LIN {X 0,Y 566.18,Z 159.454,A -85,B 0,C 180,E1 -2663.788,E2 -2663.788} C_VEL
LIN {X 0,Y 566.208,Z 159.454,A -85,B 0,C 180,E1 -2666.265,E2 -2666.265} C_VEL
LIN {X 0,Y 566.189,Z 159.457,A -85,B 0,C 180,E1 -2668.923,E2 -2668.923} C_VEL
LIN {X 0,Y 566.207,Z 159.451,A -85,B 0,C 180,E1 -2671.857,E2 -2671.857} C_VEL
LIN {X 0,Y 566.205,Z 159.457,A -85,B 0,C 180,E1 -2674.25,E2 -2674.25} C_VEL
LIN {X 0,Y 566.186,Z 159.457,A -85,B 0,C 180,E1 -2676.713,E2 -2676.713} C_VEL
LIN {X 0,Y 566.207,Z 159.452,A -85,B 0,C 180,E1 -2679.662,E2 -2679.662} C_VEL
LIN {X 0,Y 566.194,Z 159.455,A -85,B 0,C 180,E1 -2682.668,E2 -2682.668} C_VEL
LIN {X 0,Y 566.228,Z 159.45,A -85,B 0,C 180,E1 -2685.626,E2 -2685.626} C_VEL
LIN {X 0,Y 566.229,Z 159.449,A -85,B 0,C 180,E1 -2688.675,E2 -2688.675} C_VEL
LIN {X 0,Y 566.228,Z 159.45,A -85,B 0,C 180,E1 -2691.434,E2 -2691.434} C_VEL
LIN {X 0,Y 566.248,Z 159.448,A -85,B 0,C 180,E1 -2694.301,E2 -2694.301} C_VEL
LIN {X 0,Y 566.27,Z 159.45,A -85,B 0,C 180,E1 -2697.866,E2 -2697.866} C_VEL
LIN {X 0,Y 566.295,Z 159.439,A -85,B 0,C 180,E1 -2700.711,E2 -2700.711} C_VEL
LIN {X 0,Y 566.266,Z 159.444,A -85,B 0,C 180,E1 -2702.845,E2 -2702.845} C_VEL
LIN {X 0,Y 566.252,Z 159.451,A -85,B 0,C 180,E1 -2705.698,E2 -2705.698} C_VEL
LIN {X 0,Y 566.226,Z 159.448,A -85,B 0,C 180,E1 -2708.565,E2 -2708.565} C_VEL
LIN {X 0,Y 566.235,Z 159.455,A -85,B 0,C 180,E1 -2711.454,E2 -2711.454} C_VEL
LIN {X 0,Y 566.227,Z 159.449,A -85,B 0,C 180,E1 -2714.506,E2 -2714.506} C_VEL
LIN {X 0,Y 566.193,Z 159.459,A -85,B 0,C 180,E1 -2717.331,E2 -2717.331} C_VEL
LIN {X 0,Y 566.212,Z 159.45,A -85,B 0,C 180,E1 -2720.337,E2 -2720.337} C_VEL
LIN {X 0,Y 566.182,Z 159.457,A -85,B 0,C 180,E1 -2723.404,E2 -2723.404} C_VEL
LIN {X 0,Y 566.206,Z 159.451,A -85,B 0,C 180,E1 -2725.749,E2 -2725.749} C_VEL
LIN {X 0,Y 566.205,Z 159.452,A -85,B 0,C 180,E1 -2727.482,E2 -2727.482} C_VEL
LIN {X 0,Y 565.53,Z 159.536,A -85,B 0,C 180,E1 -2728.076,E2 -2728.076} C_VEL
LIN {X 0,Y 562.668,Z 159.897,A -85,B 0,C 180,E1 -2729.039,E2 -2729.039} C_VEL
LIN {X 0,Y 560.256,Z 160.195,A -85,B 0,C 180,E1 -2729.815,E2 -2729.815} C_VEL
LIN {X 0,Y 559.225,Z 160.324,A -85,B 0,C 180,E1 -2730.414,E2 -2730.414} C_VEL
LIN {X 0,Y 559.143,Z 160.332,A -85,B 0,C 180,E1 -2730.617,E2 -2730.617} C_VEL
LIN {X 0,Y 559.158,Z 160.329,A -85,B 0,C 180,E1 -2733.575,E2 -2733.575} C_VEL
LIN {X 0,Y 559.162,Z 160.335,A -85,B 0,C 180,E1 -2736.449,E2 -2736.449} C_VEL
LIN {X 0,Y 559.172,Z 160.33,A -85,B 0,C 180,E1 -2738.934,E2 -2738.934} C_VEL
LIN {X 0,Y 559.186,Z 160.326,A -85,B 0,C 180,E1 -2741.768,E2 -2741.768} C_VEL
LIN {X 0,Y 559.133,Z 160.335,A -85,B 0,C 180,E1 -2744.739,E2 -2744.739} C_VEL
LIN {X 0,Y 559.155,Z 160.329,A -85,B 0,C 180,E1 -2747.257,E2 -2747.257} C_VEL
LIN {X 0,Y 559.18,Z 160.335,A -85,B 0,C 180,E1 -2750.135,E2 -2750.135} C_VEL
LIN {X 0,Y 559.141,Z 160.331,A -85,B 0,C 180,E1 -2752.892,E2 -2752.892} C_VEL
LIN {X 0,Y 559.152,Z 160.332,A -85,B 0,C 180,E1 -2755.556,E2 -2755.556} C_VEL
LIN {X 0,Y 559.166,Z 160.334,A -85,B 0,C 180,E1 -2758.138,E2 -2758.138} C_VEL
LIN {X 0,Y 559.152,Z 160.33,A -85,B 0,C 180,E1 -2760.647,E2 -2760.647} C_VEL
LIN {X 0,Y 559.167,Z 160.329,A -85,B 0,C 180,E1 -2763.172,E2 -2763.172} C_VEL
LIN {X 0,Y 559.153,Z 160.335,A -85,B 0,C 180,E1 -2765.495,E2 -2765.495} C_VEL
LIN {X 0,Y 559.168,Z 160.327,A -85,B 0,C 180,E1 -2768.624,E2 -2768.624} C_VEL
LIN {X 0,Y 559.165,Z 160.329,A -85,B 0,C 180,E1 -2770.926,E2 -2770.926} C_VEL
LIN {X 0,Y 559.164,Z 160.332,A -85,B 0,C 180,E1 -2773.948,E2 -2773.948} C_VEL
LIN {X 0,Y 559.17,Z 160.329,A -85,B 0,C 180,E1 -2776.184,E2 -2776.184} C_VEL
LIN {X 0,Y 559.193,Z 160.332,A -85,B 0,C 180,E1 -2779.134,E2 -2779.134} C_VEL
LIN {X 0,Y 559.203,Z 160.325,A -85,B 0,C 180,E1 -2782.054,E2 -2782.054} C_VEL
LIN {X 0,Y 559.253,Z 160.324,A -85,B 0,C 180,E1 -2784.953,E2 -2784.953} C_VEL
LIN {X 0,Y 559.254,Z 160.318,A -85,B 0,C 180,E1 -2787.839,E2 -2787.839} C_VEL
LIN {X 0,Y 559.27,Z 160.322,A -85,B 0,C 180,E1 -2790.72,E2 -2790.72} C_VEL
LIN {X 0,Y 559.236,Z 160.328,A -85,B 0,C 180,E1 -2792.881,E2 -2792.881} C_VEL
LIN {X 0,Y 559.235,Z 160.32,A -85,B 0,C 180,E1 -2795.77,E2 -2795.77} C_VEL
LIN {X 0,Y 559.189,Z 160.334,A -85,B 0,C 180,E1 -2798.674,E2 -2798.674} C_VEL
LIN {X 0,Y 559.202,Z 160.324,A -85,B 0,C 180,E1 -2801.6,E2 -2801.6} C_VEL
LIN {X 0,Y 559.196,Z 160.333,A -85,B 0,C 180,E1 -2804.595,E2 -2804.595} C_VEL
LIN {X 0,Y 559.156,Z 160.33,A -85,B 0,C 180,E1 -2807.557,E2 -2807.557} C_VEL
LIN {X 0,Y 559.169,Z 160.329,A -85,B 0,C 180,E1 -2809.837,E2 -2809.837} C_VEL
LIN {X 0,Y 559.138,Z 160.338,A -85,B 0,C 180,E1 -2812.153,E2 -2812.153} C_VEL
LIN {X 0,Y 559.175,Z 160.326,A -85,B 0,C 180,E1 -2815.187,E2 -2815.187} C_VEL
LIN {X 0,Y 559.188,Z 160.328,A -85,B 0,C 180,E1 -2817.711,E2 -2817.711} C_VEL
LIN {X 0,Y 559.164,Z 160.336,A -85,B 0,C 180,E1 -2820.182,E2 -2820.182} C_VEL
LIN {X 0,Y 559.17,Z 160.328,A -85,B 0,C 180,E1 -2822.714,E2 -2822.714} C_VEL
LIN {X 0,Y 559.153,Z 160.33,A -85,B 0,C 180,E1 -2825.322,E2 -2825.322} C_VEL
LIN {X 0,Y 559.13,Z 160.339,A -85,B 0,C 180,E1 -2828.017,E2 -2828.017} C_VEL
LIN {X 0,Y 559.171,Z 160.327,A -85,B 0,C 180,E1 -2830.81,E2 -2830.81} C_VEL
LIN {X 0,Y 559.153,Z 160.338,A -85,B 0,C 180,E1 -2833.732,E2 -2833.732} C_VEL
LIN {X 0,Y 559.143,Z 160.331,A -85,B 0,C 180,E1 -2836.803,E2 -2836.803} C_VEL
LIN {X 0,Y 559.17,Z 160.331,A -85,B 0,C 180,E1 -2839.189,E2 -2839.189} C_VEL
LIN {X 0,Y 559.128,Z 160.334,A -85,B 0,C 180,E1 -2841.983,E2 -2841.983} C_VEL
LIN {X 0,Y 559.153,Z 160.331,A -85,B 0,C 180,E1 -2844.783,E2 -2844.783} C_VEL
LIN {X 0,Y 559.167,Z 160.336,A -85,B 0,C 180,E1 -2847.361,E2 -2847.361} C_VEL
LIN {X 0,Y 559.182,Z 160.326,A -85,B 0,C 180,E1 -2850.135,E2 -2850.135} C_VEL
LIN {X 0,Y 559.164,Z 160.337,A -85,B 0,C 180,E1 -2853.172,E2 -2853.172} C_VEL
LIN {X 0,Y 559.15,Z 160.333,A -85,B 0,C 180,E1 -2855.495,E2 -2855.495} C_VEL
LIN {X 0,Y 559.17,Z 160.331,A -85,B 0,C 180,E1 -2858.624,E2 -2858.624} C_VEL
LIN {X 0,Y 559.162,Z 160.337,A -85,B 0,C 180,E1 -2860.926,E2 -2860.926} C_VEL
LIN {X 0,Y 559.164,Z 160.328,A -85,B 0,C 180,E1 -2863.948,E2 -2863.948} C_VEL
LIN {X 0,Y 559.168,Z 160.329,A -85,B 0,C 180,E1 -2866.184,E2 -2866.184} C_VEL
LIN {X 0,Y 559.188,Z 160.327,A -85,B 0,C 180,E1 -2869.134,E2 -2869.134} C_VEL
LIN {X 0,Y 559.2,Z 160.326,A -85,B 0,C 180,E1 -2872.054,E2 -2872.054} C_VEL
LIN {X 0,Y 559.247,Z 160.32,A -85,B 0,C 180,E1 -2874.954,E2 -2874.954} C_VEL
LIN {X 0,Y 559.241,Z 160.32,A -85,B 0,C 180,E1 -2877.84,E2 -2877.84} C_VEL
LIN {X 0,Y 559.27,Z 160.318,A -85,B 0,C 180,E1 -2880.72,E2 -2880.72} C_VEL
LIN {X 0,Y 559.234,Z 160.32,A -85,B 0,C 180,E1 -2882.882,E2 -2882.882} C_VEL
LIN {X 0,Y 559.218,Z 160.325,A -85,B 0,C 180,E1 -2885.771,E2 -2885.771} C_VEL
LIN {X 0,Y 559.186,Z 160.326,A -85,B 0,C 180,E1 -2888.675,E2 -2888.675} C_VEL
LIN {X 0,Y 559.199,Z 160.327,A -85,B 0,C 180,E1 -2891.601,E2 -2891.601} C_VEL
LIN {X 0,Y 559.194,Z 160.325,A -85,B 0,C 180,E1 -2894.596,E2 -2894.596} C_VEL
LIN {X 0,Y 559.153,Z 160.335,A -85,B 0,C 180,E1 -2897.557,E2 -2897.557} C_VEL
LIN {X 0,Y 559.164,Z 160.335,A -85,B 0,C 180,E1 -2899.838,E2 -2899.838} C_VEL
LIN {X 0,Y 559.136,Z 160.334,A -85,B 0,C 180,E1 -2902.153,E2 -2902.153} C_VEL
LIN {X 0,Y 559.17,Z 160.332,A -85,B 0,C 180,E1 -2905.299,E2 -2905.299} C_VEL
LIN {X 0,Y 559.145,Z 160.336,A -85,B 0,C 180,E1 -2907.714,E2 -2907.714} C_VEL
LIN {X 0,Y 559.15,Z 160.33,A -85,B 0,C 180,E1 -2910.183,E2 -2910.183} C_VEL
LIN {X 0,Y 559.152,Z 160.331,A -85,B 0,C 180,E1 -2912.716,E2 -2912.716} C_VEL
LIN {X 0,Y 559.123,Z 160.342,A -85,B 0,C 180,E1 -2915.325,E2 -2915.325} C_VEL
LIN {X 0,Y 559.129,Z 160.334,A -85,B 0,C 180,E1 -2918.018,E2 -2918.018} C_VEL
LIN {X 0,Y 559.152,Z 160.336,A -85,B 0,C 180,E1 -2920.813,E2 -2920.813} C_VEL
LIN {X 0,Y 559.134,Z 160.336,A -85,B 0,C 180,E1 -2923.735,E2 -2923.735} C_VEL
LIN {X 0,Y 559.119,Z 160.342,A -85,B 0,C 180,E1 -2926.265,E2 -2926.265} C_VEL
LIN {X 0,Y 559.534,Z 163.189,A -85,B 0,C 180,E1 -2928.264,E2 -2928.264} C_VEL
LIN {X 0,Y 559.526,Z 166.347,A -85,B 0,C 180,E1 -2930.165,E2 -2930.165} C_VEL
LIN {X 0,Y 559.373,Z 171.292,A -85,B 0,C 180,E1 -2932.91,E2 -2932.91} C_VEL
LIN {X 0,Y 559.267,Z 176.344,A -85,B 0,C 180,E1 -2935.564,E2 -2935.564} C_VEL
LIN {X 0,Y 559.205,Z 181.734,A -85,B 0,C 180,E1 -2938.14,E2 -2938.14} C_VEL
LIN {X 0,Y 559.124,Z 187.123,A -85,B 0,C 180,E1 -2940.646,E2 -2940.646} C_VEL
LIN {X 0,Y 559.091,Z 192.725,A -85,B 0,C 180,E1 -2943.189,E2 -2943.189} C_VEL
LIN {X 0,Y 559.021,Z 197.902,A -85,B 0,C 180,E1 -2945.489,E2 -2945.489} C_VEL
LIN {X 0,Y 559.005,Z 204.794,A -85,B 0,C 180,E1 -2948.491,E2 -2948.491} C_VEL
LIN {X 0,Y 558.93,Z 210.478,A -85,B 0,C 180,E1 -2950.918,E2 -2950.918} C_VEL
LIN {X 0,Y 558.881,Z 215.868,A -85,B 0,C 180,E1 -2953.189,E2 -2953.189} C_VEL
LIN {X 0,Y 558.834,Z 223.054,A -85,B 0,C 180,E1 -2956.176,E2 -2956.176} C_VEL
LIN {X 0,Y 558.829,Z 225.524,A -85,B 0,C 180,E1 -2957.194,E2 -2957.194} C_VEL
LIN {X 0,Y 559.988,Z 233.412,A -85,B 0,C 180,E1 -2957.382,E2 -2957.382} C_VEL
LIN {X 0,Y 559.865,Z 245.248,A -85,B 0,C 180,E1 -2957.729,E2 -2957.729} C_VEL
LIN {X 0,Y 559.716,Z 256.248,A -85,B 0,C 180,E1 -2958.171,E2 -2958.171} C_VEL
LIN {X 0,Y 559.532,Z 267.866,A -85,B 0,C 180,E1 -2958.779,E2 -2958.779} C_VEL
LIN {X 0,Y 559.42,Z 279.921,A -85,B 0,C 180,E1 -2959.596,E2 -2959.596} C_VEL
LIN {X 0,Y 559.242,Z 289.58,A -85,B 0,C 180,E1 -2960.415,E2 -2960.415} C_VEL
LIN {X 0,Y 559.127,Z 298.385,A -85,B 0,C 180,E1 -2961.325,E2 -2961.325} C_VEL
LIN {X 0,Y 558.996,Z 307.008,A -85,B 0,C 180,E1 -2962.414,E2 -2962.414} C_VEL
LIN {X 0,Y 558.894,Z 313.872,A -85,B 0,C 180,E1 -2963.502,E2 -2963.502} C_VEL
LIN {X 0,Y 558.868,Z 319.364,A -85,B 0,C 180,E1 -2964.588,E2 -2964.588} C_VEL
LIN {X 0,Y 558.869,Z 323.664,A -85,B 0,C 180,E1 -2965.673,E2 -2965.673} C_VEL
LIN {X 0,Y 558.836,Z 325.966,A -85,B 0,C 180,E1 -2966.395,E2 -2966.395} C_VEL
LIN {X 0,Y 558.799,Z 327.792,A -85,B 0,C 180,E1 -2967.116,E2 -2967.116} C_VEL
LIN {X 0,Y 558.745,Z 330.19,A -85,B 0,C 180,E1 -2968.559,E2 -2968.559} C_VEL
LIN {X 0,Y 558.741,Z 330.782,A -85,B 0,C 180,E1 -2969.279,E2 -2969.279} C_VEL
LIN {X 0,Y 558.741,Z 330.782,A -85,B 0,C 180,E1 -2970.721,E2 -2970.721} C_VEL
LIN {X 0,Y 558.745,Z 330.19,A -85,B 0,C 180,E1 -2971.441,E2 -2971.441} C_VEL
LIN {X 0,Y 558.799,Z 327.792,A -85,B 0,C 180,E1 -2972.884,E2 -2972.884} C_VEL
LIN {X 0,Y 558.844,Z 324.879,A -85,B 0,C 180,E1 -2973.966,E2 -2973.966} C_VEL
LIN {X 0,Y 558.798,Z 320.93,A -85,B 0,C 180,E1 -2975.051,E2 -2975.051} C_VEL
LIN {X 0,Y 558.909,Z 315.835,A -85,B 0,C 180,E1 -2976.136,E2 -2976.136} C_VEL
LIN {X 0,Y 558.974,Z 309.452,A -85,B 0,C 180,E1 -2977.223,E2 -2977.223} C_VEL
LIN {X 0,Y 559.099,Z 301.491,A -85,B 0,C 180,E1 -2978.312,E2 -2978.312} C_VEL
LIN {X 0,Y 559.207,Z 293.35,A -85,B 0,C 180,E1 -2979.221,E2 -2979.221} C_VEL
LIN {X 0,Y 559.346,Z 283.358,A -85,B 0,C 180,E1 -2980.131,E2 -2980.131} C_VEL
LIN {X 0,Y 559.457,Z 273.539,A -85,B 0,C 180,E1 -2980.861,E2 -2980.861} C_VEL
LIN {X 0,Y 559.608,Z 262.505,A -85,B 0,C 180,E1 -2981.523,E2 -2981.523} C_VEL
LIN {X 0,Y 559.807,Z 248.984,A -85,B 0,C 180,E1 -2982.139,E2 -2982.139} C_VEL
LIN {X 0,Y 559.952,Z 236.981,A -85,B 0,C 180,E1 -2982.527,E2 -2982.527} C_VEL
LIN {X 0,Y 559.759,Z 231.126,A -85,B 0,C 180,E1 -2982.678,E2 -2982.678} C_VEL
LIN {X 0,Y 558.829,Z 225.524,A -85,B 0,C 180,E1 -2982.806,E2 -2982.806} C_VEL
LIN {X 0,Y 558.857,Z 219.461,A -85,B 0,C 180,E1 -2985.313,E2 -2985.313} C_VEL
LIN {X 0,Y 558.904,Z 212.275,A -85,B 0,C 180,E1 -2988.322,E2 -2988.322} C_VEL
LIN {X 0,Y 558.945,Z 206.885,A -85,B 0,C 180,E1 -2990.613,E2 -2990.613} C_VEL
LIN {X 0,Y 559.028,Z 200.432,A -85,B 0,C 180,E1 -2993.401,E2 -2993.401} C_VEL
LIN {X 0,Y 559.068,Z 194.309,A -85,B 0,C 180,E1 -2996.102,E2 -2996.102} C_VEL
LIN {X 0,Y 559.11,Z 188.92,A -85,B 0,C 180,E1 -2998.532,E2 -2998.532} C_VEL
LIN {X 0,Y 559.183,Z 182.972,A -85,B 0,C 180,E1 -3001.279,E2 -3001.279} C_VEL
LIN {X 0,Y 559.26,Z 177.321,A -85,B 0,C 180,E1 -3003.963,E2 -3003.963} C_VEL
LIN {X 0,Y 559.361,Z 172.43,A -85,B 0,C 180,E1 -3006.474,E2 -3006.474} C_VEL
LIN {X 0,Y 559.508,Z 167.979,A -85,B 0,C 180,E1 -3008.906,E2 -3008.906} C_VEL
LIN {X 0,Y 559.596,Z 164.18,A -85,B 0,C 180,E1 -3011.101,E2 -3011.101} C_VEL
LIN {X 0,Y 559.206,Z 160.915,A -85,B 0,C 180,E1 -3013.203,E2 -3013.203} C_VEL
LIN {X 0,Y 559.119,Z 160.34,A -85,B 0,C 180,E1 -3013.735,E2 -3013.735} C_VEL
LIN {X 0,Y 559.134,Z 160.335,A -85,B 0,C 180,E1 -3016.265,E2 -3016.265} C_VEL
LIN {X 0,Y 559.152,Z 160.336,A -85,B 0,C 180,E1 -3019.187,E2 -3019.187} C_VEL
LIN {X 0,Y 559.129,Z 160.334,A -85,B 0,C 180,E1 -3021.982,E2 -3021.982} C_VEL
LIN {X 0,Y 559.127,Z 160.342,A -85,B 0,C 180,E1 -3024.787,E2 -3024.787} C_VEL
LIN {X 0,Y 559.152,Z 160.33,A -85,B 0,C 180,E1 -3027.364,E2 -3027.364} C_VEL
LIN {X 0,Y 559.144,Z 160.333,A -85,B 0,C 180,E1 -3030.142,E2 -3030.142} C_VEL
LIN {X 0,Y 559.161,Z 160.329,A -85,B 0,C 180,E1 -3033.173,E2 -3033.173} C_VEL
LIN {X 0,Y 559.153,Z 160.329,A -85,B 0,C 180,E1 -3035.494,E2 -3035.494} C_VEL
LIN {X 0,Y 559.167,Z 160.332,A -85,B 0,C 180,E1 -3038.623,E2 -3038.623} C_VEL
LIN {X 0,Y 559.157,Z 160.33,A -85,B 0,C 180,E1 -3040.925,E2 -3040.925} C_VEL
LIN {X 0,Y 559.162,Z 160.334,A -85,B 0,C 180,E1 -3043.947,E2 -3043.947} C_VEL
LIN {X 0,Y 559.166,Z 160.336,A -85,B 0,C 180,E1 -3046.184,E2 -3046.184} C_VEL
LIN {X 0,Y 559.19,Z 160.325,A -85,B 0,C 180,E1 -3049.133,E2 -3049.133} C_VEL
LIN {X 0,Y 559.196,Z 160.331,A -85,B 0,C 180,E1 -3052.053,E2 -3052.053} C_VEL
LIN {X 0,Y 559.248,Z 160.317,A -85,B 0,C 180,E1 -3054.953,E2 -3054.953} C_VEL
LIN {X 0,Y 559.242,Z 160.326,A -85,B 0,C 180,E1 -3057.839,E2 -3057.839} C_VEL
LIN {X 0,Y 559.265,Z 160.315,A -85,B 0,C 180,E1 -3060.72,E2 -3060.72} C_VEL
LIN {X 0,Y 559.233,Z 160.32,A -85,B 0,C 180,E1 -3062.881,E2 -3062.881} C_VEL
LIN {X 0,Y 559.221,Z 160.326,A -85,B 0,C 180,E1 -3065.77,E2 -3065.77} C_VEL
LIN {X 0,Y 559.185,Z 160.326,A -85,B 0,C 180,E1 -3068.674,E2 -3068.674} C_VEL
LIN {X 0,Y 559.198,Z 160.329,A -85,B 0,C 180,E1 -3071.6,E2 -3071.6} C_VEL
LIN {X 0,Y 559.193,Z 160.325,A -85,B 0,C 180,E1 -3074.595,E2 -3074.595} C_VEL
LIN {X 0,Y 559.153,Z 160.333,A -85,B 0,C 180,E1 -3077.557,E2 -3077.557} C_VEL
LIN {X 0,Y 559.168,Z 160.328,A -85,B 0,C 180,E1 -3079.837,E2 -3079.837} C_VEL
LIN {X 0,Y 559.135,Z 160.331,A -85,B 0,C 180,E1 -3082.153,E2 -3082.153} C_VEL
LIN {X 0,Y 559.172,Z 160.332,A -85,B 0,C 180,E1 -3085.187,E2 -3085.187} C_VEL
LIN {X 0,Y 559.185,Z 160.325,A -85,B 0,C 180,E1 -3087.711,E2 -3087.711} C_VEL
LIN {X 0,Y 559.143,Z 160.332,A -85,B 0,C 180,E1 -3090.617,E2 -3090.617} C_VEL
LIN {X 0,Y 558.478,Z 160.418,A -85,B 0,C 180,E1 -3091.218,E2 -3091.218} C_VEL
LIN {X 0,Y 555.615,Z 160.773,A -85,B 0,C 180,E1 -3092.194,E2 -3092.194} C_VEL
LIN {X 0,Y 553.203,Z 161.075,A -85,B 0,C 180,E1 -3092.98,E2 -3092.98} C_VEL
LIN {X 0,Y 552.183,Z 161.198,A -85,B 0,C 180,E1 -3093.587,E2 -3093.587} C_VEL
LIN {X 0,Y 552.108,Z 161.207,A -85,B 0,C 180,E1 -3093.792,E2 -3093.792} C_VEL
LIN {X 0,Y 552.105,Z 161.214,A -85,B 0,C 180,E1 -3096.747,E2 -3096.747} C_VEL
LIN {X 0,Y 552.128,Z 161.204,A -85,B 0,C 180,E1 -3099.527,E2 -3099.527} C_VEL
LIN {X 0,Y 552.124,Z 161.214,A -85,B 0,C 180,E1 -3102.425,E2 -3102.425} C_VEL
LIN {X 0,Y 552.091,Z 161.209,A -85,B 0,C 180,E1 -3105.563,E2 -3105.563} C_VEL
LIN {X 0,Y 552.134,Z 161.207,A -85,B 0,C 180,E1 -3108.676,E2 -3108.676} C_VEL
LIN {X 0,Y 552.114,Z 161.207,A -85,B 0,C 180,E1 -3111.411,E2 -3111.411} C_VEL
LIN {X 0,Y 552.109,Z 161.215,A -85,B 0,C 180,E1 -3114.159,E2 -3114.159} C_VEL
LIN {X 0,Y 552.118,Z 161.206,A -85,B 0,C 180,E1 -3116.815,E2 -3116.815} C_VEL
LIN {X 0,Y 552.109,Z 161.209,A -85,B 0,C 180,E1 -3119.392,E2 -3119.392} C_VEL
LIN {X 0,Y 552.122,Z 161.214,A -85,B 0,C 180,E1 -3121.903,E2 -3121.903} C_VEL
LIN {X 0,Y 552.151,Z 161.201,A -85,B 0,C 180,E1 -3124.65,E2 -3124.65} C_VEL
LIN {X 0,Y 552.092,Z 161.216,A -85,B 0,C 180,E1 -3127.549,E2 -3127.549} C_VEL
LIN {X 0,Y 552.145,Z 161.203,A -85,B 0,C 180,E1 -3130.374,E2 -3130.374} C_VEL
LIN {X 0,Y 552.152,Z 161.205,A -85,B 0,C 180,E1 -3132.977,E2 -3132.977} C_VEL
LIN {X 0,Y 552.133,Z 161.207,A -85,B 0,C 180,E1 -3136.005,E2 -3136.005} C_VEL
LIN {X 0,Y 552.16,Z 161.206,A -85,B 0,C 180,E1 -3138.994,E2 -3138.994} C_VEL
LIN {X 0,Y 552.157,Z 161.203,A -85,B 0,C 180,E1 -3141.952,E2 -3141.952} C_VEL
LIN {X 0,Y 552.228,Z 161.198,A -85,B 0,C 180,E1 -3144.889,E2 -3144.889} C_VEL
LIN {X 0,Y 552.225,Z 161.194,A -85,B 0,C 180,E1 -3147.812,E2 -3147.812} C_VEL
LIN {X 0,Y 552.24,Z 161.198,A -85,B 0,C 180,E1 -3150.729,E2 -3150.729} C_VEL
LIN {X 0,Y 552.203,Z 161.204,A -85,B 0,C 180,E1 -3152.918,E2 -3152.918} C_VEL
LIN {X 0,Y 552.205,Z 161.196,A -85,B 0,C 180,E1 -3155.844,E2 -3155.844} C_VEL
LIN {X 0,Y 552.159,Z 161.21,A -85,B 0,C 180,E1 -3158.786,E2 -3158.786} C_VEL
LIN {X 0,Y 552.16,Z 161.201,A -85,B 0,C 180,E1 -3161.75,E2 -3161.75} C_VEL
LIN {X 0,Y 552.133,Z 161.211,A -85,B 0,C 180,E1 -3164.748,E2 -3164.748} C_VEL
LIN {X 0,Y 552.108,Z 161.209,A -85,B 0,C 180,E1 -3167.788,E2 -3167.788} C_VEL
LIN {X 0,Y 552.128,Z 161.209,A -85,B 0,C 180,E1 -3170.101,E2 -3170.101} C_VEL
LIN {X 0,Y 552.092,Z 161.216,A -85,B 0,C 180,E1 -3172.451,E2 -3172.451} C_VEL
LIN {X 0,Y 552.151,Z 161.201,A -85,B 0,C 180,E1 -3175.35,E2 -3175.35} C_VEL
LIN {X 0,Y 552.122,Z 161.214,A -85,B 0,C 180,E1 -3178.097,E2 -3178.097} C_VEL
LIN {X 0,Y 552.109,Z 161.209,A -85,B 0,C 180,E1 -3180.608,E2 -3180.608} C_VEL
LIN {X 0,Y 552.118,Z 161.206,A -85,B 0,C 180,E1 -3183.185,E2 -3183.185} C_VEL
LIN {X 0,Y 552.109,Z 161.215,A -85,B 0,C 180,E1 -3185.841,E2 -3185.841} C_VEL
LIN {X 0,Y 552.121,Z 161.206,A -85,B 0,C 180,E1 -3189.062,E2 -3189.062} C_VEL
LIN {X 0,Y 552.134,Z 161.208,A -85,B 0,C 180,E1 -3191.444,E2 -3191.444} C_VEL
LIN {X 0,Y 552.088,Z 161.209,A -85,B 0,C 180,E1 -3194.532,E2 -3194.532} C_VEL
LIN {X 0,Y 552.124,Z 161.214,A -85,B 0,C 180,E1 -3197.584,E2 -3197.584} C_VEL
LIN {X 0,Y 552.128,Z 161.204,A -85,B 0,C 180,E1 -3200.473,E2 -3200.473} C_VEL
LIN {X 0,Y 552.108,Z 161.215,A -85,B 0,C 180,E1 -3203.316,E2 -3203.316} C_VEL
LIN {X 0,Y 552.125,Z 161.206,A -85,B 0,C 180,E1 -3205.94,E2 -3205.94} C_VEL
LIN {X 0,Y 552.112,Z 161.207,A -85,B 0,C 180,E1 -3208.541,E2 -3208.541} C_VEL
LIN {X 0,Y 552.12,Z 161.211,A -85,B 0,C 180,E1 -3211.437,E2 -3211.437} C_VEL
LIN {X 0,Y 552.122,Z 161.206,A -85,B 0,C 180,E1 -3214.356,E2 -3214.356} C_VEL
LIN {X 0,Y 552.103,Z 161.213,A -85,B 0,C 180,E1 -3216.759,E2 -3216.759} C_VEL
LIN {X 0,Y 552.12,Z 161.212,A -85,B 0,C 180,E1 -3219.12,E2 -3219.12} C_VEL
LIN {X 0,Y 552.119,Z 161.207,A -85,B 0,C 180,E1 -3221.445,E2 -3221.445} C_VEL
LIN {X 0,Y 552.113,Z 161.206,A -85,B 0,C 180,E1 -3223.738,E2 -3223.738} C_VEL
LIN {X 0,Y 552.13,Z 161.205,A -85,B 0,C 180,E1 -3226.005,E2 -3226.005} C_VEL
LIN {X 0,Y 552.155,Z 161.205,A -85,B 0,C 180,E1 -3228.994,E2 -3228.994} C_VEL
LIN {X 0,Y 552.154,Z 161.203,A -85,B 0,C 180,E1 -3231.952,E2 -3231.952} C_VEL
LIN {X 0,Y 552.222,Z 161.196,A -85,B 0,C 180,E1 -3234.889,E2 -3234.889} C_VEL
LIN {X 0,Y 552.213,Z 161.195,A -85,B 0,C 180,E1 -3237.812,E2 -3237.812} C_VEL
LIN {X 0,Y 552.24,Z 161.193,A -85,B 0,C 180,E1 -3240.73,E2 -3240.73} C_VEL
LIN {X 0,Y 552.2,Z 161.196,A -85,B 0,C 180,E1 -3242.919,E2 -3242.919} C_VEL
LIN {X 0,Y 552.189,Z 161.202,A -85,B 0,C 180,E1 -3245.844,E2 -3245.844} C_VEL
LIN {X 0,Y 552.156,Z 161.201,A -85,B 0,C 180,E1 -3248.786,E2 -3248.786} C_VEL
LIN {X 0,Y 552.157,Z 161.207,A -85,B 0,C 180,E1 -3251.751,E2 -3251.751} C_VEL
LIN {X 0,Y 552.131,Z 161.204,A -85,B 0,C 180,E1 -3254.749,E2 -3254.749} C_VEL
LIN {X 0,Y 552.104,Z 161.217,A -85,B 0,C 180,E1 -3257.789,E2 -3257.789} C_VEL
LIN {X 0,Y 552.124,Z 161.208,A -85,B 0,C 180,E1 -3260.102,E2 -3260.102} C_VEL
LIN {X 0,Y 552.088,Z 161.21,A -85,B 0,C 180,E1 -3262.452,E2 -3262.452} C_VEL
LIN {X 0,Y 552.151,Z 161.208,A -85,B 0,C 180,E1 -3265.351,E2 -3265.351} C_VEL
LIN {X 0,Y 552.089,Z 161.21,A -85,B 0,C 180,E1 -3268.1,E2 -3268.1} C_VEL
LIN {X 0,Y 552.1,Z 161.208,A -85,B 0,C 180,E1 -3270.61,E2 -3270.61} C_VEL
LIN {X 0,Y 552.111,Z 161.214,A -85,B 0,C 180,E1 -3273.186,E2 -3273.186} C_VEL
LIN {X 0,Y 552.082,Z 161.213,A -85,B 0,C 180,E1 -3275.844,E2 -3275.844} C_VEL
LIN {X 0,Y 552.122,Z 161.214,A -85,B 0,C 180,E1 -3279.062,E2 -3279.062} C_VEL
LIN {X 0,Y 552.117,Z 161.212,A -85,B 0,C 180,E1 -3281.447,E2 -3281.447} C_VEL
LIN {X 0,Y 552.088,Z 161.217,A -85,B 0,C 180,E1 -3284.532,E2 -3284.532} C_VEL
LIN {X 0,Y 552.076,Z 161.218,A -85,B 0,C 180,E1 -3285.561,E2 -3285.561} C_VEL
LIN {X 0,Y 552.171,Z 161.904,A -85,B 0,C 180,E1 -3286.583,E2 -3286.583} C_VEL
LIN {X 0,Y 552.598,Z 165.036,A -85,B 0,C 180,E1 -3288.623,E2 -3288.623} C_VEL
LIN {X 0,Y 552.481,Z 169.791,A -85,B 0,C 180,E1 -3291.442,E2 -3291.442} C_VEL
LIN {X 0,Y 552.298,Z 175.428,A -85,B 0,C 180,E1 -3294.529,E2 -3294.529} C_VEL
LIN {X 0,Y 552.202,Z 180.598,A -85,B 0,C 180,E1 -3297.14,E2 -3297.14} C_VEL
LIN {X 0,Y 552.123,Z 187.123,A -85,B 0,C 180,E1 -3300.236,E2 -3300.236} C_VEL
LIN {X 0,Y 552.045,Z 193.165,A -85,B 0,C 180,E1 -3303.02,E2 -3303.02} C_VEL
LIN {X 0,Y 551.953,Z 199.699,A -85,B 0,C 180,E1 -3305.955,E2 -3305.955} C_VEL
LIN {X 0,Y 551.944,Z 205.159,A -85,B 0,C 180,E1 -3308.361,E2 -3308.361} C_VEL
LIN {X 0,Y 551.863,Z 210.478,A -85,B 0,C 180,E1 -3310.664,E2 -3310.664} C_VEL
LIN {X 0,Y 551.822,Z 215.868,A -85,B 0,C 180,E1 -3312.967,E2 -3312.967} C_VEL
LIN {X 0,Y 551.751,Z 223.054,A -85,B 0,C 180,E1 -3315.995,E2 -3315.995} C_VEL
LIN {X 0,Y 551.726,Z 225.524,A -85,B 0,C 180,E1 -3317.026,E2 -3317.026} C_VEL
LIN {X 0,Y 553.062,Z 234.322,A -85,B 0,C 180,E1 -3317.245,E2 -3317.245} C_VEL
LIN {X 0,Y 552.916,Z 246.399,A -85,B 0,C 180,E1 -3317.614,E2 -3317.614} C_VEL
LIN {X 0,Y 552.744,Z 257.449,A -85,B 0,C 180,E1 -3318.076,E2 -3318.076} C_VEL
LIN {X 0,Y 552.556,Z 269.322,A -85,B 0,C 180,E1 -3318.722,E2 -3318.722} C_VEL
LIN {X 0,Y 552.411,Z 281.081,A -85,B 0,C 180,E1 -3319.555,E2 -3319.555} C_VEL
LIN {X 0,Y 552.23,Z 289.578,A -85,B 0,C 180,E1 -3320.292,E2 -3320.292} C_VEL
LIN {X 0,Y 552.082,Z 298.38,A -85,B 0,C 180,E1 -3321.213,E2 -3321.213} C_VEL
LIN {X 0,Y 551.95,Z 307.009,A -85,B 0,C 180,E1 -3322.317,E2 -3322.317} C_VEL
LIN {X 0,Y 551.823,Z 313.873,A -85,B 0,C 180,E1 -3323.418,E2 -3323.418} C_VEL
LIN {X 0,Y 551.802,Z 319.364,A -85,B 0,C 180,E1 -3324.519,E2 -3324.519} C_VEL
LIN {X 0,Y 551.764,Z 323.663,A -85,B 0,C 180,E1 -3325.617,E2 -3325.617} C_VEL
LIN {X 0,Y 551.75,Z 325.967,A -85,B 0,C 180,E1 -3326.349,E2 -3326.349} C_VEL
LIN {X 0,Y 551.723,Z 327.79,A -85,B 0,C 180,E1 -3327.079,E2 -3327.079} C_VEL
LIN {X 0,Y 551.645,Z 330.19,A -85,B 0,C 180,E1 -3328.54,E2 -3328.54} C_VEL
LIN {X 0,Y 551.641,Z 330.782,A -85,B 0,C 180,E1 -3329.27,E2 -3329.27} C_VEL
LIN {X 0,Y 551.641,Z 330.782,A -85,B 0,C 180,E1 -3330.73,E2 -3330.73} C_VEL
LIN {X 0,Y 551.645,Z 330.19,A -85,B 0,C 180,E1 -3331.46,E2 -3331.46} C_VEL
LIN {X 0,Y 551.723,Z 327.79,A -85,B 0,C 180,E1 -3332.921,E2 -3332.921} C_VEL
LIN {X 0,Y 551.764,Z 324.876,A -85,B 0,C 180,E1 -3334.017,E2 -3334.017} C_VEL
LIN {X 0,Y 551.723,Z 320.925,A -85,B 0,C 180,E1 -3335.116,E2 -3335.116} C_VEL
LIN {X 0,Y 551.836,Z 316.435,A -85,B 0,C 180,E1 -3336.098,E2 -3336.098} C_VEL
LIN {X 0,Y 551.886,Z 310.597,A -85,B 0,C 180,E1 -3337.132,E2 -3337.132} C_VEL
LIN {X 0,Y 552.013,Z 302.934,A -85,B 0,C 180,E1 -3338.235,E2 -3338.235} C_VEL
LIN {X 0,Y 552.165,Z 293.351,A -85,B 0,C 180,E1 -3339.339,E2 -3339.339} C_VEL
LIN {X 0,Y 552.347,Z 283.351,A -85,B 0,C 180,E1 -3340.261,E2 -3340.261} C_VEL
LIN {X 0,Y 552.48,Z 273.531,A -85,B 0,C 180,E1 -3341,E2 -3341} C_VEL
LIN {X 0,Y 552.661,Z 261.747,A -85,B 0,C 180,E1 -3341.71,E2 -3341.71} C_VEL
LIN {X 0,Y 552.865,Z 248.971,A -85,B 0,C 180,E1 -3342.294,E2 -3342.294} C_VEL
LIN {X 0,Y 553.033,Z 236.965,A -85,B 0,C 180,E1 -3342.686,E2 -3342.686} C_VEL
LIN {X 0,Y 552.791,Z 231.792,A -85,B 0,C 180,E1 -3342.826,E2 -3342.826} C_VEL
LIN {X 0,Y 551.726,Z 225.524,A -85,B 0,C 180,E1 -3342.974,E2 -3342.974} C_VEL
LIN {X 0,Y 551.771,Z 219.461,A -85,B 0,C 180,E1 -3345.514,E2 -3345.514} C_VEL
LIN {X 0,Y 551.826,Z 214.071,A -85,B 0,C 180,E1 -3347.798,E2 -3347.798} C_VEL
LIN {X 0,Y 551.891,Z 208.682,A -85,B 0,C 180,E1 -3350.11,E2 -3350.11} C_VEL
LIN {X 0,Y 551.919,Z 203.292,A -85,B 0,C 180,E1 -3352.458,E2 -3352.458} C_VEL
LIN {X 0,Y 551.996,Z 196.853,A -85,B 0,C 180,E1 -3355.314,E2 -3355.314} C_VEL
LIN {X 0,Y 552.044,Z 190.716,A -85,B 0,C 180,E1 -3358.101,E2 -3358.101} C_VEL
LIN {X 0,Y 552.115,Z 185.327,A -85,B 0,C 180,E1 -3360.608,E2 -3360.608} C_VEL
LIN {X 0,Y 552.206,Z 179.937,A -85,B 0,C 180,E1 -3363.179,E2 -3363.179} C_VEL
LIN {X 0,Y 552.312,Z 174.768,A -85,B 0,C 180,E1 -3365.826,E2 -3365.826} C_VEL
LIN {X 0,Y 552.481,Z 169.791,A -85,B 0,C 180,E1 -3368.558,E2 -3368.558} C_VEL
LIN {X 0,Y 552.592,Z 164.961,A -85,B 0,C 180,E1 -3371.402,E2 -3371.402} C_VEL
LIN {X 0,Y 552.155,Z 161.798,A -85,B 0,C 180,E1 -3373.488,E2 -3373.488} C_VEL
LIN {X 0,Y 552.076,Z 161.218,A -85,B 0,C 180,E1 -3374.529,E2 -3374.529} C_VEL
LIN {X 0,Y 552.107,Z 161.211,A -85,B 0,C 180,E1 -3377.586,E2 -3377.586} C_VEL
LIN {X 0,Y 552.13,Z 161.21,A -85,B 0,C 180,E1 -3380.472,E2 -3380.472} C_VEL
LIN {X 0,Y 552.103,Z 161.21,A -85,B 0,C 180,E1 -3383.316,E2 -3383.316} C_VEL
LIN {X 0,Y 552.122,Z 161.205,A -85,B 0,C 180,E1 -3385.938,E2 -3385.938} C_VEL
LIN {X 0,Y 552.116,Z 161.214,A -85,B 0,C 180,E1 -3388.54,E2 -3388.54} C_VEL
LIN {X 0,Y 552.1,Z 161.208,A -85,B 0,C 180,E1 -3391.441,E2 -3391.441} C_VEL
LIN {X 0,Y 552.123,Z 161.213,A -85,B 0,C 180,E1 -3394.355,E2 -3394.355} C_VEL
LIN {X 0,Y 552.105,Z 161.211,A -85,B 0,C 180,E1 -3396.758,E2 -3396.758} C_VEL
LIN {X 0,Y 552.115,Z 161.206,A -85,B 0,C 180,E1 -3399.119,E2 -3399.119} C_VEL
LIN {X 0,Y 552.116,Z 161.206,A -85,B 0,C 180,E1 -3401.444,E2 -3401.444} C_VEL
LIN {X 0,Y 552.111,Z 161.209,A -85,B 0,C 180,E1 -3403.737,E2 -3403.737} C_VEL
LIN {X 0,Y 552.13,Z 161.212,A -85,B 0,C 180,E1 -3406.004,E2 -3406.004} C_VEL
LIN {X 0,Y 552.157,Z 161.201,A -85,B 0,C 180,E1 -3408.993,E2 -3408.993} C_VEL
LIN {X 0,Y 552.151,Z 161.211,A -85,B 0,C 180,E1 -3411.951,E2 -3411.951} C_VEL
LIN {X 0,Y 552.222,Z 161.193,A -85,B 0,C 180,E1 -3414.889,E2 -3414.889} C_VEL
LIN {X 0,Y 552.214,Z 161.202,A -85,B 0,C 180,E1 -3417.811,E2 -3417.811} C_VEL
LIN {X 0,Y 552.236,Z 161.191,A -85,B 0,C 180,E1 -3420.729,E2 -3420.729} C_VEL
LIN {X 0,Y 552.199,Z 161.196,A -85,B 0,C 180,E1 -3422.918,E2 -3422.918} C_VEL
LIN {X 0,Y 552.191,Z 161.201,A -85,B 0,C 180,E1 -3425.844,E2 -3425.844} C_VEL
LIN {X 0,Y 552.156,Z 161.202,A -85,B 0,C 180,E1 -3428.785,E2 -3428.785} C_VEL
LIN {X 0,Y 552.156,Z 161.204,A -85,B 0,C 180,E1 -3431.75,E2 -3431.75} C_VEL
LIN {X 0,Y 552.13,Z 161.206,A -85,B 0,C 180,E1 -3434.748,E2 -3434.748} C_VEL
LIN {X 0,Y 552.104,Z 161.208,A -85,B 0,C 180,E1 -3437.788,E2 -3437.788} C_VEL
LIN {X 0,Y 552.127,Z 161.204,A -85,B 0,C 180,E1 -3440.101,E2 -3440.101} C_VEL
LIN {X 0,Y 552.089,Z 161.211,A -85,B 0,C 180,E1 -3442.451,E2 -3442.451} C_VEL
LIN {X 0,Y 552.148,Z 161.205,A -85,B 0,C 180,E1 -3445.35,E2 -3445.35} C_VEL
LIN {X 0,Y 552.119,Z 161.206,A -85,B 0,C 180,E1 -3448.097,E2 -3448.097} C_VEL
LIN {X 0,Y 552.105,Z 161.214,A -85,B 0,C 180,E1 -3450.612,E2 -3450.612} C_VEL
LIN {X 0,Y 552.116,Z 161.208,A -85,B 0,C 180,E1 -3453.185,E2 -3453.185} C_VEL
LIN {X 0,Y 552.108,Z 161.207,A -85,B 0,C 180,E1 -3453.792,E2 -3453.792} C_VEL
LIN {X 0,Y 551.473,Z 161.293,A -85,B 0,C 180,E1 -3454.401,E2 -3454.401} C_VEL
LIN {X 0,Y 548.652,Z 161.645,A -85,B 0,C 180,E1 -3455.389,E2 -3455.389} C_VEL
LIN {X 0,Y 546.231,Z 161.948,A -85,B 0,C 180,E1 -3456.184,E2 -3456.184} C_VEL
LIN {X 0,Y 545.161,Z 162.079,A -85,B 0,C 180,E1 -3456.798,E2 -3456.798} C_VEL
LIN {X 0,Y 545.059,Z 162.088,A -85,B 0,C 180,E1 -3457.006,E2 -3457.006} C_VEL
LIN {X 0,Y 545.087,Z 162.086,A -85,B 0,C 180,E1 -3460.14,E2 -3460.14} C_VEL
LIN {X 0,Y 545.072,Z 162.084,A -85,B 0,C 180,E1 -3463.107,E2 -3463.107} C_VEL
LIN {X 0,Y 545.05,Z 162.094,A -85,B 0,C 180,E1 -3466.225,E2 -3466.225} C_VEL
LIN {X 0,Y 545.091,Z 162.082,A -85,B 0,C 180,E1 -3468.887,E2 -3468.887} C_VEL
LIN {X 0,Y 545.048,Z 162.09,A -85,B 0,C 180,E1 -3471.763,E2 -3471.763} C_VEL
LIN {X 0,Y 545.061,Z 162.087,A -85,B 0,C 180,E1 -3474.534,E2 -3474.534} C_VEL
LIN {X 0,Y 545.077,Z 162.083,A -85,B 0,C 180,E1 -3477.213,E2 -3477.213} C_VEL
LIN {X 0,Y 545.097,Z 162.088,A -85,B 0,C 180,E1 -3479.813,E2 -3479.813} C_VEL
LIN {X 0,Y 545.092,Z 162.081,A -85,B 0,C 180,E1 -3482.826,E2 -3482.826} C_VEL
LIN {X 0,Y 545.049,Z 162.094,A -85,B 0,C 180,E1 -3485.631,E2 -3485.631} C_VEL
LIN {X 0,Y 545.062,Z 162.085,A -85,B 0,C 180,E1 -3488.837,E2 -3488.837} C_VEL
LIN {X 0,Y 545.077,Z 162.087,A -85,B 0,C 180,E1 -3491.196,E2 -3491.196} C_VEL
LIN {X 0,Y 545.071,Z 162.093,A -85,B 0,C 180,E1 -3493.521,E2 -3493.521} C_VEL
LIN {X 0,Y 545.092,Z 162.086,A -85,B 0,C 180,E1 -3495.82,E2 -3495.82} C_VEL
LIN {X 0,Y 545.115,Z 162.082,A -85,B 0,C 180,E1 -3498.849,E2 -3498.849} C_VEL
LIN {X 0,Y 545.127,Z 162.08,A -85,B 0,C 180,E1 -3501.847,E2 -3501.847} C_VEL
LIN {X 0,Y 545.205,Z 162.072,A -85,B 0,C 180,E1 -3504.823,E2 -3504.823} C_VEL
LIN {X 0,Y 545.196,Z 162.07,A -85,B 0,C 180,E1 -3507.784,E2 -3507.784} C_VEL
LIN {X 0,Y 545.21,Z 162.074,A -85,B 0,C 180,E1 -3510.739,E2 -3510.739} C_VEL
LIN {X 0,Y 545.169,Z 162.08,A -85,B 0,C 180,E1 -3512.956,E2 -3512.956} C_VEL
LIN {X 0,Y 545.177,Z 162.072,A -85,B 0,C 180,E1 -3515.919,E2 -3515.919} C_VEL
LIN {X 0,Y 545.118,Z 162.085,A -85,B 0,C 180,E1 -3518.9,E2 -3518.9} C_VEL
LIN {X 0,Y 545.132,Z 162.078,A -85,B 0,C 180,E1 -3521.904,E2 -3521.904} C_VEL
LIN {X 0,Y 545.082,Z 162.087,A -85,B 0,C 180,E1 -3524.943,E2 -3524.943} C_VEL
LIN {X 0,Y 545.076,Z 162.087,A -85,B 0,C 180,E1 -3528.026,E2 -3528.026} C_VEL
LIN {X 0,Y 545.092,Z 162.09,A -85,B 0,C 180,E1 -3530.372,E2 -3530.372} C_VEL
LIN {X 0,Y 545.087,Z 162.082,A -85,B 0,C 180,E1 -3533.559,E2 -3533.559} C_VEL
LIN {X 0,Y 545.075,Z 162.089,A -85,B 0,C 180,E1 -3536,E2 -3536} C_VEL
LIN {X 0,Y 545.088,Z 162.083,A -85,B 0,C 180,E1 -3538.749,E2 -3538.749} C_VEL
LIN {X 0,Y 545.074,Z 162.087,A -85,B 0,C 180,E1 -3541.682,E2 -3541.682} C_VEL
LIN {X 0,Y 545.077,Z 162.084,A -85,B 0,C 180,E1 -3544.563,E2 -3544.563} C_VEL
LIN {X 0,Y 545.034,Z 162.09,A -85,B 0,C 180,E1 -3547.303,E2 -3547.303} C_VEL
LIN {X 0,Y 545.088,Z 162.085,A -85,B 0,C 180,E1 -3550.14,E2 -3550.14} C_VEL
LIN {X 0,Y 545.073,Z 162.085,A -85,B 0,C 180,E1 -3553.106,E2 -3553.106} C_VEL
LIN {X 0,Y 545.061,Z 162.086,A -85,B 0,C 180,E1 -3556.224,E2 -3556.224} C_VEL
LIN {X 0,Y 545.095,Z 162.082,A -85,B 0,C 180,E1 -3558.887,E2 -3558.887} C_VEL
LIN {X 0,Y 545.047,Z 162.091,A -85,B 0,C 180,E1 -3561.763,E2 -3561.763} C_VEL
LIN {X 0,Y 545.058,Z 162.085,A -85,B 0,C 180,E1 -3564.534,E2 -3564.534} C_VEL
LIN {X 0,Y 545.075,Z 162.091,A -85,B 0,C 180,E1 -3567.212,E2 -3567.212} C_VEL
LIN {X 0,Y 545.095,Z 162.082,A -85,B 0,C 180,E1 -3569.813,E2 -3569.813} C_VEL
LIN {X 0,Y 545.089,Z 162.086,A -85,B 0,C 180,E1 -3572.826,E2 -3572.826} C_VEL
LIN {X 0,Y 545.045,Z 162.088,A -85,B 0,C 180,E1 -3575.631,E2 -3575.631} C_VEL
LIN {X 0,Y 545.063,Z 162.092,A -85,B 0,C 180,E1 -3578.837,E2 -3578.837} C_VEL
LIN {X 0,Y 545.074,Z 162.087,A -85,B 0,C 180,E1 -3581.196,E2 -3581.196} C_VEL
LIN {X 0,Y 545.069,Z 162.084,A -85,B 0,C 180,E1 -3583.522,E2 -3583.522} C_VEL
LIN {X 0,Y 545.089,Z 162.081,A -85,B 0,C 180,E1 -3585.82,E2 -3585.82} C_VEL
LIN {X 0,Y 545.111,Z 162.085,A -85,B 0,C 180,E1 -3588.85,E2 -3588.85} C_VEL
LIN {X 0,Y 545.124,Z 162.078,A -85,B 0,C 180,E1 -3591.847,E2 -3591.847} C_VEL
LIN {X 0,Y 545.198,Z 162.072,A -85,B 0,C 180,E1 -3594.823,E2 -3594.823} C_VEL
LIN {X 0,Y 545.185,Z 162.071,A -85,B 0,C 180,E1 -3597.784,E2 -3597.784} C_VEL
LIN {X 0,Y 545.209,Z 162.069,A -85,B 0,C 180,E1 -3600.739,E2 -3600.739} C_VEL
LIN {X 0,Y 545.166,Z 162.072,A -85,B 0,C 180,E1 -3602.956,E2 -3602.956} C_VEL
LIN {X 0,Y 545.161,Z 162.078,A -85,B 0,C 180,E1 -3605.92,E2 -3605.92} C_VEL
LIN {X 0,Y 545.115,Z 162.078,A -85,B 0,C 180,E1 -3608.901,E2 -3608.901} C_VEL
LIN {X 0,Y 545.129,Z 162.085,A -85,B 0,C 180,E1 -3611.905,E2 -3611.905} C_VEL
LIN {X 0,Y 545.08,Z 162.082,A -85,B 0,C 180,E1 -3614.944,E2 -3614.944} C_VEL
LIN {X 0,Y 545.071,Z 162.089,A -85,B 0,C 180,E1 -3618.026,E2 -3618.026} C_VEL
LIN {X 0,Y 545.089,Z 162.082,A -85,B 0,C 180,E1 -3620.373,E2 -3620.373} C_VEL
LIN {X 0,Y 545.084,Z 162.091,A -85,B 0,C 180,E1 -3623.56,E2 -3623.56} C_VEL
LIN {X 0,Y 545.072,Z 162.086,A -85,B 0,C 180,E1 -3626.001,E2 -3626.001} C_VEL
LIN {X 0,Y 545.07,Z 162.084,A -85,B 0,C 180,E1 -3628.746,E2 -3628.746} C_VEL
LIN {X 0,Y 545.054,Z 162.09,A -85,B 0,C 180,E1 -3631.679,E2 -3631.679} C_VEL
LIN {X 0,Y 545.058,Z 162.087,A -85,B 0,C 180,E1 -3634.565,E2 -3634.565} C_VEL
LIN {X 0,Y 545.033,Z 162.097,A -85,B 0,C 180,E1 -3637.305,E2 -3637.305} C_VEL
LIN {X 0,Y 545.065,Z 162.087,A -85,B 0,C 180,E1 -3640.143,E2 -3640.143} C_VEL
LIN {X 0,Y 545.046,Z 162.094,A -85,B 0,C 180,E1 -3642.696,E2 -3642.696} C_VEL
LIN {X 0,Y 545.025,Z 162.097,A -85,B 0,C 180,E1 -3645.172,E2 -3645.172} C_VEL
LIN {X 0,Y 545.027,Z 162.168,A -85,B 0,C 180,E1 -3645.869,E2 -3645.869} C_VEL
LIN {X 0,Y 545.556,Z 165.856,A -85,B 0,C 180,E1 -3648.346,E2 -3648.346} C_VEL
LIN {X 0,Y 545.544,Z 169.999,A -85,B 0,C 180,E1 -3650.859,E2 -3650.859} C_VEL
LIN {X 0,Y 545.307,Z 174.922,A -85,B 0,C 180,E1 -3653.641,E2 -3653.641} C_VEL
LIN {X 0,Y 545.197,Z 179.998,A -85,B 0,C 180,E1 -3656.338,E2 -3656.338} C_VEL
LIN {X 0,Y 545.089,Z 185.327,A -85,B 0,C 180,E1 -3658.954,E2 -3658.954} C_VEL
LIN {X 0,Y 545.023,Z 190.716,A -85,B 0,C 180,E1 -3661.504,E2 -3661.504} C_VEL
LIN {X 0,Y 544.946,Z 196.106,A -85,B 0,C 180,E1 -3663.993,E2 -3663.993} C_VEL
LIN {X 0,Y 544.884,Z 201.495,A -85,B 0,C 180,E1 -3666.432,E2 -3666.432} C_VEL
LIN {X 0,Y 544.844,Z 206.885,A -85,B 0,C 180,E1 -3668.828,E2 -3668.828} C_VEL
LIN {X 0,Y 544.752,Z 212.275,A -85,B 0,C 180,E1 -3671.184,E2 -3671.184} C_VEL
LIN {X 0,Y 544.707,Z 217.664,A -85,B 0,C 180,E1 -3673.51,E2 -3673.51} C_VEL
LIN {X 0,Y 544.684,Z 223.054,A -85,B 0,C 180,E1 -3675.809,E2 -3675.809} C_VEL
LIN {X 0,Y 544.627,Z 225.524,A -85,B 0,C 180,E1 -3676.854,E2 -3676.854} C_VEL
LIN {X 0,Y 546.127,Z 235.202,A -85,B 0,C 180,E1 -3677.104,E2 -3677.104} C_VEL
LIN {X 0,Y 546,Z 246.389,A -85,B 0,C 180,E1 -3677.455,E2 -3677.455} C_VEL
LIN {X 0,Y 545.789,Z 257.445,A -85,B 0,C 180,E1 -3677.922,E2 -3677.922} C_VEL
LIN {X 0,Y 545.566,Z 269.709,A -85,B 0,C 180,E1 -3678.601,E2 -3678.601} C_VEL
LIN {X 0,Y 545.405,Z 281.08,A -85,B 0,C 180,E1 -3679.419,E2 -3679.419} C_VEL
LIN {X 0,Y 545.222,Z 289.574,A -85,B 0,C 180,E1 -3680.166,E2 -3680.166} C_VEL
LIN {X 0,Y 545.062,Z 298.376,A -85,B 0,C 180,E1 -3681.099,E2 -3681.099} C_VEL
LIN {X 0,Y 544.896,Z 307.009,A -85,B 0,C 180,E1 -3682.217,E2 -3682.217} C_VEL
LIN {X 0,Y 544.76,Z 314.282,A -85,B 0,C 180,E1 -3683.408,E2 -3683.408} C_VEL
LIN {X 0,Y 544.738,Z 319.364,A -85,B 0,C 180,E1 -3684.447,E2 -3684.447} C_VEL
LIN {X 0,Y 544.66,Z 323.661,A -85,B 0,C 180,E1 -3685.56,E2 -3685.56} C_VEL
LIN {X 0,Y 544.669,Z 325.968,A -85,B 0,C 180,E1 -3686.301,E2 -3686.301} C_VEL
LIN {X 0,Y 544.65,Z 327.787,A -85,B 0,C 180,E1 -3687.041,E2 -3687.041} C_VEL
LIN {X 0,Y 544.546,Z 330.191,A -85,B 0,C 180,E1 -3688.521,E2 -3688.521} C_VEL
LIN {X 0,Y 544.542,Z 330.781,A -85,B 0,C 180,E1 -3689.261,E2 -3689.261} C_VEL
LIN {X 0,Y 544.542,Z 330.781,A -85,B 0,C 180,E1 -3690.739,E2 -3690.739} C_VEL
LIN {X 0,Y 544.546,Z 330.191,A -85,B 0,C 180,E1 -3691.479,E2 -3691.479} C_VEL
LIN {X 0,Y 544.65,Z 327.787,A -85,B 0,C 180,E1 -3692.959,E2 -3692.959} C_VEL
LIN {X 0,Y 544.684,Z 324.872,A -85,B 0,C 180,E1 -3694.069,E2 -3694.069} C_VEL
LIN {X 0,Y 544.653,Z 320.921,A -85,B 0,C 180,E1 -3695.182,E2 -3695.182} C_VEL
LIN {X 0,Y 544.723,Z 315.628,A -85,B 0,C 180,E1 -3696.335,E2 -3696.335} C_VEL
LIN {X 0,Y 544.836,Z 309.442,A -85,B 0,C 180,E1 -3697.411,E2 -3697.411} C_VEL
LIN {X 0,Y 545.006,Z 301.494,A -85,B 0,C 180,E1 -3698.528,E2 -3698.528} C_VEL
LIN {X 0,Y 545.139,Z 293.353,A -85,B 0,C 180,E1 -3699.461,E2 -3699.461} C_VEL
LIN {X 0,Y 545.351,Z 283.345,A -85,B 0,C 180,E1 -3700.394,E2 -3700.394} C_VEL
LIN {X 0,Y 545.516,Z 273.523,A -85,B 0,C 180,E1 -3701.142,E2 -3701.142} C_VEL
LIN {X 0,Y 545.681,Z 262.711,A -85,B 0,C 180,E1 -3701.81,E2 -3701.81} C_VEL
LIN {X 0,Y 545.894,Z 250.154,A -85,B 0,C 180,E1 -3702.406,E2 -3702.406} C_VEL
LIN {X 0,Y 546.097,Z 237.823,A -85,B 0,C 180,E1 -3702.826,E2 -3702.826} C_VEL
LIN {X 0,Y 545.902,Z 232.945,A -85,B 0,C 180,E1 -3702.961,E2 -3702.961} C_VEL
LIN {X 0,Y 544.627,Z 225.524,A -85,B 0,C 180,E1 -3703.146,E2 -3703.146} C_VEL
LIN {X 0,Y 544.677,Z 221.257,A -85,B 0,C 180,E1 -3704.955,E2 -3704.955} C_VEL
LIN {X 0,Y 544.737,Z 214.071,A -85,B 0,C 180,E1 -3708.037,E2 -3708.037} C_VEL
LIN {X 0,Y 544.819,Z 208.682,A -85,B 0,C 180,E1 -3710.383,E2 -3710.383} C_VEL
LIN {X 0,Y 544.871,Z 203.292,A -85,B 0,C 180,E1 -3712.765,E2 -3712.765} C_VEL
LIN {X 0,Y 544.935,Z 197.278,A -85,B 0,C 180,E1 -3715.473,E2 -3715.473} C_VEL
LIN {X 0,Y 544.979,Z 192.513,A -85,B 0,C 180,E1 -3717.661,E2 -3717.661} C_VEL
LIN {X 0,Y 545.099,Z 186.992,A -85,B 0,C 180,E1 -3720.249,E2 -3720.249} C_VEL
LIN {X 0,Y 545.195,Z 181.151,A -85,B 0,C 180,E1 -3723.08,E2 -3723.08} C_VEL
LIN {X 0,Y 545.29,Z 176.107,A -85,B 0,C 180,E1 -3725.71,E2 -3725.71} C_VEL
LIN {X 0,Y 545.464,Z 171.601,A -85,B 0,C 180,E1 -3728.203,E2 -3728.203} C_VEL
LIN {X 0,Y 545.599,Z 166.782,A -85,B 0,C 180,E1 -3731.066,E2 -3731.066} C_VEL
LIN {X 0,Y 545.289,Z 163.692,A -85,B 0,C 180,E1 -3733.085,E2 -3733.085} C_VEL
LIN {X 0,Y 545.027,Z 162.175,A -85,B 0,C 180,E1 -3734.131,E2 -3734.131} C_VEL
LIN {X 0,Y 545.043,Z 162.095,A -85,B 0,C 180,E1 -3736.889,E2 -3736.889} C_VEL
LIN {X 0,Y 545.079,Z 162.086,A -85,B 0,C 180,E1 -3739.527,E2 -3739.527} C_VEL
LIN {X 0,Y 545.047,Z 162.088,A -85,B 0,C 180,E1 -3741.863,E2 -3741.863} C_VEL
LIN {X 0,Y 545.032,Z 162.094,A -85,B 0,C 180,E1 -3744.531,E2 -3744.531} C_VEL
LIN {X 0,Y 545.065,Z 162.086,A -85,B 0,C 180,E1 -3747.211,E2 -3747.211} C_VEL
LIN {X 0,Y 545.06,Z 162.085,A -85,B 0,C 180,E1 -3749.81,E2 -3749.81} C_VEL
LIN {X 0,Y 545.078,Z 162.087,A -85,B 0,C 180,E1 -3752.828,E2 -3752.828} C_VEL
LIN {X 0,Y 545.048,Z 162.087,A -85,B 0,C 180,E1 -3755.63,E2 -3755.63} C_VEL
LIN {X 0,Y 545.061,Z 162.087,A -85,B 0,C 180,E1 -3758.836,E2 -3758.836} C_VEL
LIN {X 0,Y 545.07,Z 162.083,A -85,B 0,C 180,E1 -3761.195,E2 -3761.195} C_VEL
LIN {X 0,Y 545.068,Z 162.085,A -85,B 0,C 180,E1 -3763.521,E2 -3763.521} C_VEL
LIN {X 0,Y 545.089,Z 162.086,A -85,B 0,C 180,E1 -3765.819,E2 -3765.819} C_VEL
LIN {X 0,Y 545.113,Z 162.078,A -85,B 0,C 180,E1 -3768.849,E2 -3768.849} C_VEL
LIN {X 0,Y 545.122,Z 162.085,A -85,B 0,C 180,E1 -3771.847,E2 -3771.847} C_VEL
LIN {X 0,Y 545.197,Z 162.068,A -85,B 0,C 180,E1 -3774.822,E2 -3774.822} C_VEL
LIN {X 0,Y 545.186,Z 162.078,A -85,B 0,C 180,E1 -3777.783,E2 -3777.783} C_VEL
LIN {X 0,Y 545.206,Z 162.067,A -85,B 0,C 180,E1 -3780.738,E2 -3780.738} C_VEL
LIN {X 0,Y 545.166,Z 162.073,A -85,B 0,C 180,E1 -3782.955,E2 -3782.955} C_VEL
LIN {X 0,Y 545.163,Z 162.075,A -85,B 0,C 180,E1 -3785.919,E2 -3785.919} C_VEL
LIN {X 0,Y 545.115,Z 162.08,A -85,B 0,C 180,E1 -3788.9,E2 -3788.9} C_VEL
LIN {X 0,Y 545.128,Z 162.078,A -85,B 0,C 180,E1 -3791.904,E2 -3791.904} C_VEL
LIN {X 0,Y 545.079,Z 162.087,A -85,B 0,C 180,E1 -3794.943,E2 -3794.943} C_VEL
LIN {X 0,Y 545.072,Z 162.083,A -85,B 0,C 180,E1 -3798.026,E2 -3798.026} C_VEL
LIN {X 0,Y 545.092,Z 162.082,A -85,B 0,C 180,E1 -3800.372,E2 -3800.372} C_VEL
LIN {X 0,Y 545.084,Z 162.083,A -85,B 0,C 180,E1 -3803.559,E2 -3803.559} C_VEL
LIN {X 0,Y 545.072,Z 162.083,A -85,B 0,C 180,E1 -3806,E2 -3806} C_VEL
LIN {X 0,Y 545.086,Z 162.09,A -85,B 0,C 180,E1 -3808.749,E2 -3808.749} C_VEL
LIN {X 0,Y 545.063,Z 162.089,A -85,B 0,C 180,E1 -3811.048,E2 -3811.048} C_VEL
LIN {X 0,Y 545.061,Z 162.085,A -85,B 0,C 180,E1 -3813.79,E2 -3813.79} C_VEL
LIN {X 0,Y 545.068,Z 162.088,A -85,B 0,C 180,E1 -3816.927,E2 -3816.927} C_VEL
LIN {X 0,Y 545.059,Z 162.088,A -85,B 0,C 180,E1 -3817.006,E2 -3817.006} C_VEL
LIN {X 0,Y 544.353,Z 162.175,A -85,B 0,C 180,E1 -3817.623,E2 -3817.623} C_VEL
LIN {X 0,Y 541.499,Z 162.536,A -85,B 0,C 180,E1 -3818.624,E2 -3818.624} C_VEL
LIN {X 0,Y 539.122,Z 162.828,A -85,B 0,C 180,E1 -3819.43,E2 -3819.43} C_VEL
LIN {X 0,Y 538.116,Z 162.953,A -85,B 0,C 180,E1 -3820.052,E2 -3820.052} C_VEL
LIN {X 0,Y 538.041,Z 162.96,A -85,B 0,C 180,E1 -3820.262,E2 -3820.262} C_VEL
LIN {X 0,Y 538.019,Z 162.963,A -85,B 0,C 180,E1 -3822.988,E2 -3822.988} C_VEL
LIN {X 0,Y 538.018,Z 162.966,A -85,B 0,C 180,E1 -3825.926,E2 -3825.926} C_VEL
LIN {X 0,Y 538.046,Z 162.958,A -85,B 0,C 180,E1 -3829.252,E2 -3829.252} C_VEL
LIN {X 0,Y 537.989,Z 162.975,A -85,B 0,C 180,E1 -3832.123,E2 -3832.123} C_VEL
LIN {X 0,Y 538.015,Z 162.962,A -85,B 0,C 180,E1 -3834.918,E2 -3834.918} C_VEL
LIN {X 0,Y 538.027,Z 162.965,A -85,B 0,C 180,E1 -3837.618,E2 -3837.618} C_VEL
LIN {X 0,Y 538.039,Z 162.963,A -85,B 0,C 180,E1 -3840.241,E2 -3840.241} C_VEL
LIN {X 0,Y 538.062,Z 162.956,A -85,B 0,C 180,E1 -3842.797,E2 -3842.797} C_VEL
LIN {X 0,Y 538.045,Z 162.962,A -85,B 0,C 180,E1 -3845.293,E2 -3845.293} C_VEL
LIN {X 0,Y 538.011,Z 162.966,A -85,B 0,C 180,E1 -3848.042,E2 -3848.042} C_VEL
LIN {X 0,Y 538.034,Z 162.961,A -85,B 0,C 180,E1 -3850.94,E2 -3850.94} C_VEL
LIN {X 0,Y 538.022,Z 162.969,A -85,B 0,C 180,E1 -3853.299,E2 -3853.299} C_VEL
LIN {X 0,Y 538.061,Z 162.964,A -85,B 0,C 180,E1 -3855.631,E2 -3855.631} C_VEL
LIN {X 0,Y 538.074,Z 162.957,A -85,B 0,C 180,E1 -3858.702,E2 -3858.702} C_VEL
LIN {X 0,Y 538.084,Z 162.958,A -85,B 0,C 180,E1 -3861.74,E2 -3861.74} C_VEL
LIN {X 0,Y 538.163,Z 162.949,A -85,B 0,C 180,E1 -3864.755,E2 -3864.755} C_VEL
LIN {X 0,Y 538.167,Z 162.946,A -85,B 0,C 180,E1 -3867.755,E2 -3867.755} C_VEL
LIN {X 0,Y 538.18,Z 162.95,A -85,B 0,C 180,E1 -3870.748,E2 -3870.748} C_VEL
LIN {X 0,Y 538.136,Z 162.956,A -85,B 0,C 180,E1 -3872.994,E2 -3872.994} C_VEL
LIN {X 0,Y 538.131,Z 162.95,A -85,B 0,C 180,E1 -3875.997,E2 -3875.997} C_VEL
LIN {X 0,Y 538.069,Z 162.962,A -85,B 0,C 180,E1 -3879.017,E2 -3879.017} C_VEL
LIN {X 0,Y 538.08,Z 162.957,A -85,B 0,C 180,E1 -3882.062,E2 -3882.062} C_VEL
LIN {X 0,Y 538.042,Z 162.962,A -85,B 0,C 180,E1 -3885.144,E2 -3885.144} C_VEL
LIN {X 0,Y 538.028,Z 162.969,A -85,B 0,C 180,E1 -3888.27,E2 -3888.27} C_VEL
LIN {X 0,Y 538.036,Z 162.965,A -85,B 0,C 180,E1 -3890.651,E2 -3890.651} C_VEL
LIN {X 0,Y 538.02,Z 162.965,A -85,B 0,C 180,E1 -3893.887,E2 -3893.887} C_VEL
LIN {X 0,Y 538.038,Z 162.966,A -85,B 0,C 180,E1 -3896.366,E2 -3896.366} C_VEL
LIN {X 0,Y 538.052,Z 162.958,A -85,B 0,C 180,E1 -3898.938,E2 -3898.938} C_VEL
LIN {X 0,Y 538.023,Z 162.968,A -85,B 0,C 180,E1 -3901.89,E2 -3901.89} C_VEL
LIN {X 0,Y 538.027,Z 162.962,A -85,B 0,C 180,E1 -3904.621,E2 -3904.621} C_VEL
LIN {X 0,Y 538.003,Z 162.965,A -85,B 0,C 180,E1 -3907.17,E2 -3907.17} C_VEL
LIN {X 0,Y 538.049,Z 162.967,A -85,B 0,C 180,E1 -3909.794,E2 -3909.794} C_VEL
LIN {X 0,Y 538.013,Z 162.963,A -85,B 0,C 180,E1 -3912.786,E2 -3912.786} C_VEL
LIN {X 0,Y 538.024,Z 162.966,A -85,B 0,C 180,E1 -3915.925,E2 -3915.925} C_VEL
LIN {X 0,Y 538.072,Z 162.96,A -85,B 0,C 180,E1 -3919.249,E2 -3919.249} C_VEL
LIN {X 0,Y 537.987,Z 162.967,A -85,B 0,C 180,E1 -3922.122,E2 -3922.122} C_VEL
LIN {X 0,Y 538.013,Z 162.965,A -85,B 0,C 180,E1 -3924.917,E2 -3924.917} C_VEL
LIN {X 0,Y 538.019,Z 162.966,A -85,B 0,C 180,E1 -3927.618,E2 -3927.618} C_VEL
LIN {X 0,Y 538.036,Z 162.96,A -85,B 0,C 180,E1 -3930.241,E2 -3930.241} C_VEL
LIN {X 0,Y 538.059,Z 162.961,A -85,B 0,C 180,E1 -3932.796,E2 -3932.796} C_VEL
LIN {X 0,Y 538.042,Z 162.965,A -85,B 0,C 180,E1 -3935.293,E2 -3935.293} C_VEL
LIN {X 0,Y 538.008,Z 162.963,A -85,B 0,C 180,E1 -3938.042,E2 -3938.042} C_VEL
LIN {X 0,Y 538.032,Z 162.969,A -85,B 0,C 180,E1 -3940.94,E2 -3940.94} C_VEL
LIN {X 0,Y 538.02,Z 162.964,A -85,B 0,C 180,E1 -3943.299,E2 -3943.299} C_VEL
LIN {X 0,Y 538.057,Z 162.957,A -85,B 0,C 180,E1 -3945.631,E2 -3945.631} C_VEL
LIN {X 0,Y 538.07,Z 162.964,A -85,B 0,C 180,E1 -3948.702,E2 -3948.702} C_VEL
LIN {X 0,Y 538.081,Z 162.954,A -85,B 0,C 180,E1 -3951.74,E2 -3951.74} C_VEL
LIN {X 0,Y 538.155,Z 162.95,A -85,B 0,C 180,E1 -3954.755,E2 -3954.755} C_VEL
LIN {X 0,Y 538.158,Z 162.946,A -85,B 0,C 180,E1 -3957.755,E2 -3957.755} C_VEL
LIN {X 0,Y 538.179,Z 162.945,A -85,B 0,C 180,E1 -3960.749,E2 -3960.749} C_VEL
LIN {X 0,Y 538.133,Z 162.948,A -85,B 0,C 180,E1 -3962.995,E2 -3962.995} C_VEL
LIN {X 0,Y 538.115,Z 162.957,A -85,B 0,C 180,E1 -3965.998,E2 -3965.998} C_VEL
LIN {X 0,Y 538.065,Z 162.956,A -85,B 0,C 180,E1 -3969.018,E2 -3969.018} C_VEL
LIN {X 0,Y 538.077,Z 162.962,A -85,B 0,C 180,E1 -3972.063,E2 -3972.063} C_VEL
LIN {X 0,Y 538.04,Z 162.96,A -85,B 0,C 180,E1 -3975.144,E2 -3975.144} C_VEL
LIN {X 0,Y 538.024,Z 162.964,A -85,B 0,C 180,E1 -3978.271,E2 -3978.271} C_VEL
LIN {X 0,Y 538.034,Z 162.96,A -85,B 0,C 180,E1 -3980.652,E2 -3980.652} C_VEL
LIN {X 0,Y 538.02,Z 162.967,A -85,B 0,C 180,E1 -3983.888,E2 -3983.888} C_VEL
LIN {X 0,Y 538.034,Z 162.96,A -85,B 0,C 180,E1 -3986.367,E2 -3986.367} C_VEL
LIN {X 0,Y 538.026,Z 162.963,A -85,B 0,C 180,E1 -3988.934,E2 -3988.934} C_VEL
LIN {X 0,Y 538.006,Z 162.966,A -85,B 0,C 180,E1 -3991.888,E2 -3991.888} C_VEL
LIN {X 0,Y 538.008,Z 162.966,A -85,B 0,C 180,E1 -3994.618,E2 -3994.618} C_VEL
LIN {X 0,Y 538.001,Z 162.973,A -85,B 0,C 180,E1 -3997.171,E2 -3997.171} C_VEL
LIN {X 0,Y 538.022,Z 162.965,A -85,B 0,C 180,E1 -3999.797,E2 -3999.797} C_VEL
LIN {X 0,Y 537.998,Z 162.973,A -85,B 0,C 180,E1 -4002.789,E2 -4002.789} C_VEL
LIN {X 0,Y 537.998,Z 162.973,A -85,B 0,C 180,E1 -4005.138,E2 -4005.138} C_VEL
LIN {X 0,Y 538.136,Z 163.946,A -85,B 0,C 180,E1 -4006.198,E2 -4006.198} C_VEL
LIN {X 0,Y 538.583,Z 167.004,A -85,B 0,C 180,E1 -4008.28,E2 -4008.28} C_VEL
LIN {X 0,Y 538.507,Z 171.796,A -85,B 0,C 180,E1 -4011.213,E2 -4011.213} C_VEL
LIN {X 0,Y 538.298,Z 176.783,A -85,B 0,C 180,E1 -4014.045,E2 -4014.045} C_VEL
LIN {X 0,Y 538.165,Z 181.83,A -85,B 0,C 180,E1 -4016.737,E2 -4016.737} C_VEL
LIN {X 0,Y 538.044,Z 187.493,A -85,B 0,C 180,E1 -4019.554,E2 -4019.554} C_VEL
LIN {X 0,Y 537.958,Z 192.513,A -85,B 0,C 180,E1 -4021.946,E2 -4021.946} C_VEL
LIN {X 0,Y 537.875,Z 197.902,A -85,B 0,C 180,E1 -4024.458,E2 -4024.458} C_VEL
LIN {X 0,Y 537.798,Z 203.292,A -85,B 0,C 180,E1 -4026.919,E2 -4026.919} C_VEL
LIN {X 0,Y 537.756,Z 208.682,A -85,B 0,C 180,E1 -4029.338,E2 -4029.338} C_VEL
LIN {X 0,Y 537.663,Z 214.071,A -85,B 0,C 180,E1 -4031.717,E2 -4031.717} C_VEL
LIN {X 0,Y 537.617,Z 219.461,A -85,B 0,C 180,E1 -4034.067,E2 -4034.067} C_VEL
LIN {X 0,Y 537.571,Z 225.524,A -85,B 0,C 180,E1 -4036.678,E2 -4036.678} C_VEL
LIN {X 0,Y 539.218,Z 236.06,A -85,B 0,C 180,E1 -4036.959,E2 -4036.959} C_VEL
LIN {X 0,Y 539.048,Z 247.666,A -85,B 0,C 180,E1 -4037.338,E2 -4037.338} C_VEL
LIN {X 0,Y 538.815,Z 259.409,A -85,B 0,C 180,E1 -4037.859,E2 -4037.859} C_VEL
LIN {X 0,Y 538.55,Z 271.842,A -85,B 0,C 180,E1 -4038.594,E2 -4038.594} C_VEL
LIN {X 0,Y 538.389,Z 282.207,A -85,B 0,C 180,E1 -4039.375,E2 -4039.375} C_VEL
LIN {X 0,Y 538.133,Z 291.481,A -85,B 0,C 180,E1 -4040.225,E2 -4040.225} C_VEL
LIN {X 0,Y 537.979,Z 299.991,A -85,B 0,C 180,E1 -4041.17,E2 -4041.17} C_VEL
LIN {X 0,Y 537.817,Z 308.25,A -85,B 0,C 180,E1 -4042.303,E2 -4042.303} C_VEL
LIN {X 0,Y 537.697,Z 314.686,A -85,B 0,C 180,E1 -4043.397,E2 -4043.397} C_VEL
LIN {X 0,Y 537.673,Z 319.363,A -85,B 0,C 180,E1 -4044.374,E2 -4044.374} C_VEL
LIN {X 0,Y 537.557,Z 323.659,A -85,B 0,C 180,E1 -4045.501,E2 -4045.501} C_VEL
LIN {X 0,Y 537.591,Z 325.97,A -85,B 0,C 180,E1 -4046.252,E2 -4046.252} C_VEL
LIN {X 0,Y 537.551,Z 327.785,A -85,B 0,C 180,E1 -4047.002,E2 -4047.002} C_VEL
LIN {X 0,Y 537.451,Z 330.192,A -85,B 0,C 180,E1 -4048.501,E2 -4048.501} C_VEL
LIN {X 0,Y 537.442,Z 330.781,A -85,B 0,C 180,E1 -4049.251,E2 -4049.251} C_VEL
LIN {X 0,Y 537.442,Z 330.781,A -85,B 0,C 180,E1 -4050.749,E2 -4050.749} C_VEL
LIN {X 0,Y 537.451,Z 330.192,A -85,B 0,C 180,E1 -4051.499,E2 -4051.499} C_VEL
LIN {X 0,Y 537.551,Z 327.785,A -85,B 0,C 180,E1 -4052.998,E2 -4052.998} C_VEL
LIN {X 0,Y 537.603,Z 324.869,A -85,B 0,C 180,E1 -4054.123,E2 -4054.123} C_VEL
LIN {X 0,Y 537.587,Z 320.917,A -85,B 0,C 180,E1 -4055.251,E2 -4055.251} C_VEL
LIN {X 0,Y 537.638,Z 316.123,A -85,B 0,C 180,E1 -4056.32,E2 -4056.32} C_VEL
LIN {X 0,Y 537.754,Z 310.588,A -85,B 0,C 180,E1 -4057.321,E2 -4057.321} C_VEL
LIN {X 0,Y 537.883,Z 304.296,A -85,B 0,C 180,E1 -4058.263,E2 -4058.263} C_VEL
LIN {X 0,Y 538.052,Z 296.751,A -85,B 0,C 180,E1 -4059.207,E2 -4059.207} C_VEL
LIN {X 0,Y 538.22,Z 287.634,A -85,B 0,C 180,E1 -4060.153,E2 -4060.153} C_VEL
LIN {X 0,Y 538.475,Z 276.208,A -85,B 0,C 180,E1 -4061.099,E2 -4061.099} C_VEL
LIN {X 0,Y 538.659,Z 265.075,A -85,B 0,C 180,E1 -4061.827,E2 -4061.827} C_VEL
LIN {X 0,Y 538.886,Z 253.425,A -85,B 0,C 180,E1 -4062.426,E2 -4062.426} C_VEL
LIN {X 0,Y 539.179,Z 239.511,A -85,B 0,C 180,E1 -4062.946,E2 -4062.946} C_VEL
LIN {X 0,Y 538.971,Z 233.855,A -85,B 0,C 180,E1 -4063.107,E2 -4063.107} C_VEL
LIN {X 0,Y 537.571,Z 225.524,A -85,B 0,C 180,E1 -4063.322,E2 -4063.322} C_VEL
LIN {X 0,Y 537.617,Z 219.461,A -85,B 0,C 180,E1 -4065.933,E2 -4065.933} C_VEL
LIN {X 0,Y 537.661,Z 214.071,A -85,B 0,C 180,E1 -4068.283,E2 -4068.283} C_VEL
LIN {X 0,Y 537.756,Z 208.682,A -85,B 0,C 180,E1 -4070.662,E2 -4070.662} C_VEL
LIN {X 0,Y 537.798,Z 203.292,A -85,B 0,C 180,E1 -4073.081,E2 -4073.081} C_VEL
LIN {X 0,Y 537.883,Z 197.699,A -85,B 0,C 180,E1 -4075.636,E2 -4075.636} C_VEL
LIN {X 0,Y 537.958,Z 192.513,A -85,B 0,C 180,E1 -4078.054,E2 -4078.054} C_VEL
LIN {X 0,Y 538.039,Z 187.123,A -85,B 0,C 180,E1 -4080.625,E2 -4080.625} C_VEL
LIN {X 0,Y 538.165,Z 181.754,A -85,B 0,C 180,E1 -4083.301,E2 -4083.301} C_VEL
LIN {X 0,Y 538.299,Z 176.738,A -85,B 0,C 180,E1 -4085.98,E2 -4085.98} C_VEL
LIN {X 0,Y 538.507,Z 171.775,A -85,B 0,C 180,E1 -4088.787,E2 -4088.787} C_VEL
LIN {X 0,Y 538.6,Z 168.423,A -85,B 0,C 180,E1 -4090.815,E2 -4090.815} C_VEL
LIN {X 0,Y 538.338,Z 165.062,A -85,B 0,C 180,E1 -4093.023,E2 -4093.023} C_VEL
LIN {X 0,Y 538.078,Z 163.542,A -85,B 0,C 180,E1 -4094.079,E2 -4094.079} C_VEL
LIN {X 0,Y 538,Z 162.971,A -85,B 0,C 180,E1 -4095.137,E2 -4095.137} C_VEL
LIN {X 0,Y 538.021,Z 162.966,A -85,B 0,C 180,E1 -4098.225,E2 -4098.225} C_VEL
LIN {X 0,Y 538.011,Z 162.969,A -85,B 0,C 180,E1 -4101.169,E2 -4101.169} C_VEL
LIN {X 0,Y 537.991,Z 162.967,A -85,B 0,C 180,E1 -4104.088,E2 -4104.088} C_VEL
LIN {X 0,Y 538.027,Z 162.97,A -85,B 0,C 180,E1 -4106.727,E2 -4106.727} C_VEL
LIN {X 0,Y 538.023,Z 162.961,A -85,B 0,C 180,E1 -4109.556,E2 -4109.556} C_VEL
LIN {X 0,Y 538.042,Z 162.966,A -85,B 0,C 180,E1 -4112.65,E2 -4112.65} C_VEL
LIN {X 0,Y 538.045,Z 162.959,A -85,B 0,C 180,E1 -4115.292,E2 -4115.292} C_VEL
LIN {X 0,Y 538.011,Z 162.968,A -85,B 0,C 180,E1 -4118.041,E2 -4118.041} C_VEL
LIN {X 0,Y 538.028,Z 162.962,A -85,B 0,C 180,E1 -4120.939,E2 -4120.939} C_VEL
LIN {X 0,Y 538.019,Z 162.962,A -85,B 0,C 180,E1 -4123.298,E2 -4123.298} C_VEL
LIN {X 0,Y 538.058,Z 162.96,A -85,B 0,C 180,E1 -4125.63,E2 -4125.63} C_VEL
LIN {X 0,Y 538.072,Z 162.956,A -85,B 0,C 180,E1 -4128.701,E2 -4128.701} C_VEL
LIN {X 0,Y 538.08,Z 162.961,A -85,B 0,C 180,E1 -4131.739,E2 -4131.739} C_VEL
LIN {X 0,Y 538.155,Z 162.945,A -85,B 0,C 180,E1 -4134.755,E2 -4134.755} C_VEL
LIN {X 0,Y 538.159,Z 162.954,A -85,B 0,C 180,E1 -4137.754,E2 -4137.754} C_VEL
LIN {X 0,Y 538.176,Z 162.942,A -85,B 0,C 180,E1 -4140.748,E2 -4140.748} C_VEL
LIN {X 0,Y 538.133,Z 162.949,A -85,B 0,C 180,E1 -4142.994,E2 -4142.994} C_VEL
LIN {X 0,Y 538.116,Z 162.952,A -85,B 0,C 180,E1 -4145.997,E2 -4145.997} C_VEL
LIN {X 0,Y 538.065,Z 162.96,A -85,B 0,C 180,E1 -4149.017,E2 -4149.017} C_VEL
LIN {X 0,Y 538.077,Z 162.955,A -85,B 0,C 180,E1 -4152.062,E2 -4152.062} C_VEL
LIN {X 0,Y 538.039,Z 162.967,A -85,B 0,C 180,E1 -4155.143,E2 -4155.143} C_VEL
LIN {X 0,Y 538.025,Z 162.961,A -85,B 0,C 180,E1 -4158.27,E2 -4158.27} C_VEL
LIN {X 0,Y 538.036,Z 162.963,A -85,B 0,C 180,E1 -4160.651,E2 -4160.651} C_VEL
LIN {X 0,Y 538.017,Z 162.962,A -85,B 0,C 180,E1 -4163.887,E2 -4163.887} C_VEL
LIN {X 0,Y 538.035,Z 162.962,A -85,B 0,C 180,E1 -4166.367,E2 -4166.367} C_VEL
LIN {X 0,Y 538.05,Z 162.966,A -85,B 0,C 180,E1 -4168.939,E2 -4168.939} C_VEL
LIN {X 0,Y 538.007,Z 162.964,A -85,B 0,C 180,E1 -4171.888,E2 -4171.888} C_VEL
LIN {X 0,Y 538.025,Z 162.97,A -85,B 0,C 180,E1 -4174.621,E2 -4174.621} C_VEL
LIN {X 0,Y 538.001,Z 162.966,A -85,B 0,C 180,E1 -4177.171,E2 -4177.171} C_VEL
LIN {X 0,Y 538.041,Z 162.96,A -85,B 0,C 180,E1 -4180.262,E2 -4180.262} C_VEL
LIN {X 0,Y 537.389,Z 163.045,A -85,B 0,C 180,E1 -4180.887,E2 -4180.887} C_VEL
LIN {X 0,Y 534.528,Z 163.399,A -85,B 0,C 180,E1 -4181.902,E2 -4181.902} C_VEL
LIN {X 0,Y 532.095,Z 163.704,A -85,B 0,C 180,E1 -4182.718,E2 -4182.718} C_VEL
LIN {X 0,Y 531.044,Z 163.831,A -85,B 0,C 180,E1 -4183.349,E2 -4183.349} C_VEL
LIN {X 0,Y 530.956,Z 163.842,A -85,B 0,C 180,E1 -4183.563,E2 -4183.563} C_VEL
LIN {X 0,Y 530.953,Z 163.848,A -85,B 0,C 180,E1 -4186.505,E2 -4186.505} C_VEL
LIN {X 0,Y 530.983,Z 163.839,A -85,B 0,C 180,E1 -4188.976,E2 -4188.976} C_VEL
LIN {X 0,Y 530.954,Z 163.843,A -85,B 0,C 180,E1 -4191.53,E2 -4191.53} C_VEL
LIN {X 0,Y 530.977,Z 163.843,A -85,B 0,C 180,E1 -4194.382,E2 -4194.382} C_VEL
LIN {X 0,Y 530.968,Z 163.84,A -85,B 0,C 180,E1 -4197.134,E2 -4197.134} C_VEL
LIN {X 0,Y 530.982,Z 163.846,A -85,B 0,C 180,E1 -4199.804,E2 -4199.804} C_VEL
LIN {X 0,Y 531.012,Z 163.836,A -85,B 0,C 180,E1 -4202.467,E2 -4202.467} C_VEL
LIN {X 0,Y 531.002,Z 163.836,A -85,B 0,C 180,E1 -4204.943,E2 -4204.943} C_VEL
LIN {X 0,Y 530.967,Z 163.842,A -85,B 0,C 180,E1 -4208.247,E2 -4208.247} C_VEL
LIN {X 0,Y 530.992,Z 163.837,A -85,B 0,C 180,E1 -4210.678,E2 -4210.678} C_VEL
LIN {X 0,Y 530.983,Z 163.843,A -85,B 0,C 180,E1 -4213.071,E2 -4213.071} C_VEL
LIN {X 0,Y 531.037,Z 163.841,A -85,B 0,C 180,E1 -4215.437,E2 -4215.437} C_VEL
LIN {X 0,Y 531.034,Z 163.834,A -85,B 0,C 180,E1 -4218.55,E2 -4218.55} C_VEL
LIN {X 0,Y 531.054,Z 163.835,A -85,B 0,C 180,E1 -4221.63,E2 -4221.63} C_VEL
LIN {X 0,Y 531.122,Z 163.825,A -85,B 0,C 180,E1 -4224.685,E2 -4224.685} C_VEL
LIN {X 0,Y 531.139,Z 163.822,A -85,B 0,C 180,E1 -4227.725,E2 -4227.725} C_VEL
LIN {X 0,Y 531.15,Z 163.825,A -85,B 0,C 180,E1 -4230.758,E2 -4230.758} C_VEL
LIN {X 0,Y 531.103,Z 163.832,A -85,B 0,C 180,E1 -4233.034,E2 -4233.034} C_VEL
LIN {X 0,Y 531.089,Z 163.827,A -85,B 0,C 180,E1 -4236.077,E2 -4236.077} C_VEL
LIN {X 0,Y 531.029,Z 163.838,A -85,B 0,C 180,E1 -4239.138,E2 -4239.138} C_VEL
LIN {X 0,Y 531.038,Z 163.836,A -85,B 0,C 180,E1 -4242.225,E2 -4242.225} C_VEL
LIN {X 0,Y 530.992,Z 163.839,A -85,B 0,C 180,E1 -4245.35,E2 -4245.35} C_VEL
LIN {X 0,Y 530.987,Z 163.847,A -85,B 0,C 180,E1 -4248.521,E2 -4248.521} C_VEL
LIN {X 0,Y 530.996,Z 163.839,A -85,B 0,C 180,E1 -4250.938,E2 -4250.938} C_VEL
LIN {X 0,Y 530.976,Z 163.848,A -85,B 0,C 180,E1 -4254.224,E2 -4254.224} C_VEL
LIN {X 0,Y 531.002,Z 163.838,A -85,B 0,C 180,E1 -4256.743,E2 -4256.743} C_VEL
LIN {X 0,Y 530.996,Z 163.837,A -85,B 0,C 180,E1 -4259.321,E2 -4259.321} C_VEL
LIN {X 0,Y 530.976,Z 163.848,A -85,B 0,C 180,E1 -4262.103,E2 -4262.103} C_VEL
LIN {X 0,Y 530.984,Z 163.838,A -85,B 0,C 180,E1 -4264.854,E2 -4264.854} C_VEL
LIN {X 0,Y 530.961,Z 163.845,A -85,B 0,C 180,E1 -4267.507,E2 -4267.507} C_VEL
LIN {X 0,Y 531.003,Z 163.837,A -85,B 0,C 180,E1 -4270.43,E2 -4270.43} C_VEL
LIN {X 0,Y 530.953,Z 163.848,A -85,B 0,C 180,E1 -4273.495,E2 -4273.495} C_VEL
LIN {X 0,Y 530.958,Z 163.842,A -85,B 0,C 180,E1 -4276.505,E2 -4276.505} C_VEL
LIN {X 0,Y 531.02,Z 163.842,A -85,B 0,C 180,E1 -4279.571,E2 -4279.571} C_VEL
LIN {X 0,Y 530.962,Z 163.841,A -85,B 0,C 180,E1 -4282.577,E2 -4282.577} C_VEL
LIN {X 0,Y 530.995,Z 163.846,A -85,B 0,C 180,E1 -4285.311,E2 -4285.311} C_VEL
LIN {X 0,Y 530.964,Z 163.841,A -85,B 0,C 180,E1 -4288.032,E2 -4288.032} C_VEL
LIN {X 0,Y 531.001,Z 163.841,A -85,B 0,C 180,E1 -4290.871,E2 -4290.871} C_VEL
LIN {X 0,Y 530.999,Z 163.843,A -85,B 0,C 180,E1 -4293.257,E2 -4293.257} C_VEL
LIN {X 0,Y 530.99,Z 163.837,A -85,B 0,C 180,E1 -4295.958,E2 -4295.958} C_VEL
LIN {X 0,Y 530.996,Z 163.844,A -85,B 0,C 180,E1 -4299.062,E2 -4299.062} C_VEL
LIN {X 0,Y 531.01,Z 163.837,A -85,B 0,C 180,E1 -4302.278,E2 -4302.278} C_VEL
LIN {X 0,Y 531.012,Z 163.836,A -85,B 0,C 180,E1 -4305.436,E2 -4305.436} C_VEL
LIN {X 0,Y 531.03,Z 163.84,A -85,B 0,C 180,E1 -4308.55,E2 -4308.55} C_VEL
LIN {X 0,Y 531.05,Z 163.83,A -85,B 0,C 180,E1 -4311.63,E2 -4311.63} C_VEL
LIN {X 0,Y 531.114,Z 163.828,A -85,B 0,C 180,E1 -4314.686,E2 -4314.686} C_VEL
LIN {X 0,Y 531.13,Z 163.821,A -85,B 0,C 180,E1 -4317.725,E2 -4317.725} C_VEL
LIN {X 0,Y 531.149,Z 163.82,A -85,B 0,C 180,E1 -4320.759,E2 -4320.759} C_VEL
LIN {X 0,Y 531.099,Z 163.824,A -85,B 0,C 180,E1 -4323.035,E2 -4323.035} C_VEL
LIN {X 0,Y 531.075,Z 163.835,A -85,B 0,C 180,E1 -4326.078,E2 -4326.078} C_VEL
LIN {X 0,Y 531.025,Z 163.833,A -85,B 0,C 180,E1 -4329.139,E2 -4329.139} C_VEL
LIN {X 0,Y 531.035,Z 163.837,A -85,B 0,C 180,E1 -4332.225,E2 -4332.225} C_VEL
LIN {X 0,Y 530.99,Z 163.84,A -85,B 0,C 180,E1 -4335.35,E2 -4335.35} C_VEL
LIN {X 0,Y 530.983,Z 163.839,A -85,B 0,C 180,E1 -4338.522,E2 -4338.522} C_VEL
LIN {X 0,Y 530.995,Z 163.837,A -85,B 0,C 180,E1 -4340.939,E2 -4340.939} C_VEL
LIN {X 0,Y 530.976,Z 163.84,A -85,B 0,C 180,E1 -4344.225,E2 -4344.225} C_VEL
LIN {X 0,Y 530.993,Z 163.838,A -85,B 0,C 180,E1 -4346.745,E2 -4346.745} C_VEL
LIN {X 0,Y 530.976,Z 163.847,A -85,B 0,C 180,E1 -4349.323,E2 -4349.323} C_VEL
LIN {X 0,Y 530.962,Z 163.842,A -85,B 0,C 180,E1 -4352.101,E2 -4352.101} C_VEL
LIN {X 0,Y 530.966,Z 163.845,A -85,B 0,C 180,E1 -4354.852,E2 -4354.852} C_VEL
LIN {X 0,Y 530.962,Z 163.848,A -85,B 0,C 180,E1 -4357.508,E2 -4357.508} C_VEL
LIN {X 0,Y 530.979,Z 163.843,A -85,B 0,C 180,E1 -4360.434,E2 -4360.434} C_VEL
LIN {X 0,Y 530.942,Z 163.851,A -85,B 0,C 180,E1 -4363.497,E2 -4363.497} C_VEL
LIN {X 0,Y 530.97,Z 163.848,A -85,B 0,C 180,E1 -4364.549,E2 -4364.549} C_VEL
LIN {X 0,Y 531.034,Z 164.414,A -85,B 0,C 180,E1 -4365.616,E2 -4365.616} C_VEL
LIN {X 0,Y 531.511,Z 167.496,A -85,B 0,C 180,E1 -4367.772,E2 -4367.772} C_VEL
LIN {X 0,Y 531.562,Z 171.089,A -85,B 0,C 180,E1 -4370.072,E2 -4370.072} C_VEL
LIN {X 0,Y 531.384,Z 175.227,A -85,B 0,C 180,E1 -4372.528,E2 -4372.528} C_VEL
LIN {X 0,Y 531.198,Z 180.22,A -85,B 0,C 180,E1 -4375.326,E2 -4375.326} C_VEL
LIN {X 0,Y 531.091,Z 185.418,A -85,B 0,C 180,E1 -4378.041,E2 -4378.041} C_VEL
LIN {X 0,Y 530.967,Z 191.135,A -85,B 0,C 180,E1 -4380.879,E2 -4380.879} C_VEL
LIN {X 0,Y 530.847,Z 197.902,A -85,B 0,C 180,E1 -4384.095,E2 -4384.095} C_VEL
LIN {X 0,Y 530.741,Z 203.292,A -85,B 0,C 180,E1 -4386.594,E2 -4386.594} C_VEL
LIN {X 0,Y 530.711,Z 208.682,A -85,B 0,C 180,E1 -4389.051,E2 -4389.051} C_VEL
LIN {X 0,Y 530.588,Z 214.071,A -85,B 0,C 180,E1 -4391.465,E2 -4391.465} C_VEL
LIN {X 0,Y 530.531,Z 219.461,A -85,B 0,C 180,E1 -4393.848,E2 -4393.848} C_VEL
LIN {X 0,Y 530.49,Z 225.299,A -85,B 0,C 180,E1 -4396.4,E2 -4396.4} C_VEL
LIN {X 0,Y 530.471,Z 225.524,A -85,B 0,C 180,E1 -4396.497,E2 -4396.497} C_VEL
LIN {X 0,Y 532.296,Z 236.918,A -85,B 0,C 180,E1 -4396.811,E2 -4396.811} C_VEL
LIN {X 0,Y 532.112,Z 248.942,A -85,B 0,C 180,E1 -4397.219,E2 -4397.219} C_VEL
LIN {X 0,Y 531.833,Z 261.201,A -85,B 0,C 180,E1 -4397.794,E2 -4397.794} C_VEL
LIN {X 0,Y 531.587,Z 272.043,A -85,B 0,C 180,E1 -4398.457,E2 -4398.457} C_VEL
LIN {X 0,Y 531.368,Z 282.201,A -85,B 0,C 180,E1 -4399.233,E2 -4399.233} C_VEL
LIN {X 0,Y 531.108,Z 291.476,A -85,B 0,C 180,E1 -4400.095,E2 -4400.095} C_VEL
LIN {X 0,Y 530.94,Z 299.988,A -85,B 0,C 180,E1 -4401.052,E2 -4401.052} C_VEL
LIN {X 0,Y 530.758,Z 308.251,A -85,B 0,C 180,E1 -4402.2,E2 -4402.2} C_VEL
LIN {X 0,Y 530.596,Z 315.247,A -85,B 0,C 180,E1 -4403.421,E2 -4403.421} C_VEL
LIN {X 0,Y 530.523,Z 320.912,A -85,B 0,C 180,E1 -4404.679,E2 -4404.679} C_VEL
LIN {X 0,Y 530.522,Z 324.865,A -85,B 0,C 180,E1 -4405.822,E2 -4405.822} C_VEL
LIN {X 0,Y 530.457,Z 327.782,A -85,B 0,C 180,E1 -4406.962,E2 -4406.962} C_VEL
LIN {X 0,Y 530.361,Z 330.193,A -85,B 0,C 180,E1 -4408.481,E2 -4408.481} C_VEL
LIN {X 0,Y 530.344,Z 330.781,A -85,B 0,C 180,E1 -4409.241,E2 -4409.241} C_VEL
LIN {X 0,Y 530.344,Z 330.781,A -85,B 0,C 180,E1 -4410.759,E2 -4410.759} C_VEL
LIN {X 0,Y 530.361,Z 330.193,A -85,B 0,C 180,E1 -4411.519,E2 -4411.519} C_VEL
LIN {X 0,Y 530.457,Z 327.782,A -85,B 0,C 180,E1 -4413.038,E2 -4413.038} C_VEL
LIN {X 0,Y 530.522,Z 324.865,A -85,B 0,C 180,E1 -4414.178,E2 -4414.178} C_VEL
LIN {X 0,Y 530.523,Z 320.912,A -85,B 0,C 180,E1 -4415.321,E2 -4415.321} C_VEL
LIN {X 0,Y 530.593,Z 315.262,A -85,B 0,C 180,E1 -4416.575,E2 -4416.575} C_VEL
LIN {X 0,Y 530.758,Z 308.251,A -85,B 0,C 180,E1 -4417.8,E2 -4417.8} C_VEL
LIN {X 0,Y 530.94,Z 299.988,A -85,B 0,C 180,E1 -4418.948,E2 -4418.948} C_VEL
LIN {X 0,Y 531.109,Z 291.476,A -85,B 0,C 180,E1 -4419.905,E2 -4419.905} C_VEL
LIN {X 0,Y 531.354,Z 282.201,A -85,B 0,C 180,E1 -4420.767,E2 -4420.767} C_VEL
LIN {X 0,Y 531.601,Z 272.072,A -85,B 0,C 180,E1 -4421.541,E2 -4421.541} C_VEL
LIN {X 0,Y 531.786,Z 261.201,A -85,B 0,C 180,E1 -4422.207,E2 -4422.207} C_VEL
LIN {X 0,Y 532.082,Z 248.942,A -85,B 0,C 180,E1 -4422.782,E2 -4422.782} C_VEL
LIN {X 0,Y 532.288,Z 236.918,A -85,B 0,C 180,E1 -4423.189,E2 -4423.189} C_VEL
LIN {X 0,Y 530.471,Z 225.524,A -85,B 0,C 180,E1 -4423.503,E2 -4423.503} C_VEL
LIN {X 0,Y 530.523,Z 221.257,A -85,B 0,C 180,E1 -4425.363,E2 -4425.363} C_VEL
LIN {X 0,Y 530.594,Z 215.868,A -85,B 0,C 180,E1 -4427.737,E2 -4427.737} C_VEL
LIN {X 0,Y 530.684,Z 210.478,A -85,B 0,C 180,E1 -4430.14,E2 -4430.14} C_VEL
LIN {X 0,Y 530.736,Z 205.089,A -85,B 0,C 180,E1 -4432.582,E2 -4432.582} C_VEL
LIN {X 0,Y 530.788,Z 199.699,A -85,B 0,C 180,E1 -4435.068,E2 -4435.068} C_VEL
LIN {X 0,Y 530.895,Z 194.309,A -85,B 0,C 180,E1 -4437.602,E2 -4437.602} C_VEL
LIN {X 0,Y 530.986,Z 188.931,A -85,B 0,C 180,E1 -4440.195,E2 -4440.195} C_VEL
LIN {X 0,Y 531.11,Z 183.663,A -85,B 0,C 180,E1 -4442.856,E2 -4442.856} C_VEL
LIN {X 0,Y 531.261,Z 178.554,A -85,B 0,C 180,E1 -4445.596,E2 -4445.596} C_VEL
LIN {X 0,Y 531.495,Z 173.057,A -85,B 0,C 180,E1 -4448.724,E2 -4448.724} C_VEL
LIN {X 0,Y 531.603,Z 168.771,A -85,B 0,C 180,E1 -4451.377,E2 -4451.377} C_VEL
LIN {X 0,Y 531.23,Z 165.693,A -85,B 0,C 180,E1 -4453.467,E2 -4453.467} C_VEL
LIN {X 0,Y 530.986,Z 164.179,A -85,B 0,C 180,E1 -4454.546,E2 -4454.546} C_VEL
LIN {X 0,Y 530.942,Z 163.85,A -85,B 0,C 180,E1 -4456.503,E2 -4456.503} C_VEL
LIN {X 0,Y 530.979,Z 163.843,A -85,B 0,C 180,E1 -4459.566,E2 -4459.566} C_VEL
LIN {X 0,Y 530.965,Z 163.848,A -85,B 0,C 180,E1 -4462.576,E2 -4462.576} C_VEL
LIN {X 0,Y 530.978,Z 163.841,A -85,B 0,C 180,E1 -4465.309,E2 -4465.309} C_VEL
LIN {X 0,Y 530.963,Z 163.842,A -85,B 0,C 180,E1 -4468.031,E2 -4468.031} C_VEL
LIN {X 0,Y 530.984,Z 163.843,A -85,B 0,C 180,E1 -4470.874,E2 -4470.874} C_VEL
LIN {X 0,Y 530.993,Z 163.838,A -85,B 0,C 180,E1 -4473.255,E2 -4473.255} C_VEL
LIN {X 0,Y 530.993,Z 163.84,A -85,B 0,C 180,E1 -4475.957,E2 -4475.957} C_VEL
LIN {X 0,Y 530.995,Z 163.837,A -85,B 0,C 180,E1 -4479.061,E2 -4479.061} C_VEL
LIN {X 0,Y 531.011,Z 163.843,A -85,B 0,C 180,E1 -4482.277,E2 -4482.277} C_VEL
LIN {X 0,Y 531.014,Z 163.835,A -85,B 0,C 180,E1 -4485.435,E2 -4485.435} C_VEL
LIN {X 0,Y 531.031,Z 163.834,A -85,B 0,C 180,E1 -4488.549,E2 -4488.549} C_VEL
LIN {X 0,Y 531.05,Z 163.835,A -85,B 0,C 180,E1 -4491.629,E2 -4491.629} C_VEL
LIN {X 0,Y 531.114,Z 163.822,A -85,B 0,C 180,E1 -4494.685,E2 -4494.685} C_VEL
LIN {X 0,Y 531.131,Z 163.829,A -85,B 0,C 180,E1 -4497.725,E2 -4497.725} C_VEL
LIN {X 0,Y 531.146,Z 163.818,A -85,B 0,C 180,E1 -4500.758,E2 -4500.758} C_VEL
LIN {X 0,Y 531.099,Z 163.826,A -85,B 0,C 180,E1 -4503.034,E2 -4503.034} C_VEL
LIN {X 0,Y 531.076,Z 163.828,A -85,B 0,C 180,E1 -4506.077,E2 -4506.077} C_VEL
LIN {X 0,Y 531.025,Z 163.838,A -85,B 0,C 180,E1 -4509.138,E2 -4509.138} C_VEL
LIN {X 0,Y 531.034,Z 163.832,A -85,B 0,C 180,E1 -4512.225,E2 -4512.225} C_VEL
LIN {X 0,Y 530.989,Z 163.845,A -85,B 0,C 180,E1 -4515.349,E2 -4515.349} C_VEL
LIN {X 0,Y 530.984,Z 163.84,A -85,B 0,C 180,E1 -4518.521,E2 -4518.521} C_VEL
LIN {X 0,Y 530.996,Z 163.844,A -85,B 0,C 180,E1 -4520.938,E2 -4520.938} C_VEL
LIN {X 0,Y 530.973,Z 163.84,A -85,B 0,C 180,E1 -4524.224,E2 -4524.224} C_VEL
LIN {X 0,Y 530.999,Z 163.843,A -85,B 0,C 180,E1 -4526.743,E2 -4526.743} C_VEL
LIN {X 0,Y 530.994,Z 163.839,A -85,B 0,C 180,E1 -4529.321,E2 -4529.321} C_VEL
LIN {X 0,Y 530.963,Z 163.842,A -85,B 0,C 180,E1 -4532.101,E2 -4532.101} C_VEL
LIN {X 0,Y 530.982,Z 163.844,A -85,B 0,C 180,E1 -4534.854,E2 -4534.854} C_VEL
LIN {X 0,Y 530.96,Z 163.841,A -85,B 0,C 180,E1 -4537.508,E2 -4537.508} C_VEL
LIN {X 0,Y 531.02,Z 163.842,A -85,B 0,C 180,E1 -4540.429,E2 -4540.429} C_VEL
LIN {X 0,Y 530.956,Z 163.842,A -85,B 0,C 180,E1 -4543.563,E2 -4543.563} C_VEL
LIN {X 0,Y 530.283,Z 163.933,A -85,B 0,C 180,E1 -4544.197,E2 -4544.197} C_VEL
LIN {X 0,Y 527.432,Z 164.286,A -85,B 0,C 180,E1 -4545.225,E2 -4545.225} C_VEL
LIN {X 0,Y 525.028,Z 164.586,A -85,B 0,C 180,E1 -4546.054,E2 -4546.054} C_VEL
LIN {X 0,Y 523.995,Z 164.713,A -85,B 0,C 180,E1 -4546.693,E2 -4546.693} C_VEL
LIN {X 0,Y 523.911,Z 164.721,A -85,B 0,C 180,E1 -4546.91,E2 -4546.91} C_VEL
LIN {X 0,Y 523.938,Z 164.717,A -85,B 0,C 180,E1 -4548.908,E2 -4548.908} C_VEL
LIN {X 0,Y 523.911,Z 164.725,A -85,B 0,C 180,E1 -4551.899,E2 -4551.899} C_VEL
LIN {X 0,Y 523.934,Z 164.717,A -85,B 0,C 180,E1 -4554.909,E2 -4554.909} C_VEL
LIN {X 0,Y 523.938,Z 164.721,A -85,B 0,C 180,E1 -4557.678,E2 -4557.678} C_VEL
LIN {X 0,Y 523.965,Z 164.713,A -85,B 0,C 180,E1 -4560.673,E2 -4560.673} C_VEL
LIN {X 0,Y 523.971,Z 164.72,A -85,B 0,C 180,E1 -4563.729,E2 -4563.729} C_VEL
LIN {X 0,Y 523.932,Z 164.718,A -85,B 0,C 180,E1 -4566.271,E2 -4566.271} C_VEL
LIN {X 0,Y 523.942,Z 164.716,A -85,B 0,C 180,E1 -4568.767,E2 -4568.767} C_VEL
LIN {X 0,Y 523.948,Z 164.719,A -85,B 0,C 180,E1 -4571.221,E2 -4571.221} C_VEL
LIN {X 0,Y 523.934,Z 164.724,A -85,B 0,C 180,E1 -4573.639,E2 -4573.639} C_VEL
LIN {X 0,Y 523.942,Z 164.719,A -85,B 0,C 180,E1 -4576.028,E2 -4576.028} C_VEL
LIN {X 0,Y 524.009,Z 164.709,A -85,B 0,C 180,E1 -4578.394,E2 -4578.394} C_VEL
LIN {X 0,Y 524.002,Z 164.715,A -85,B 0,C 180,E1 -4581.516,E2 -4581.516} C_VEL
LIN {X 0,Y 524.084,Z 164.702,A -85,B 0,C 180,E1 -4584.614,E2 -4584.614} C_VEL
LIN {X 0,Y 524.111,Z 164.697,A -85,B 0,C 180,E1 -4587.695,E2 -4587.695} C_VEL
LIN {X 0,Y 524.121,Z 164.701,A -85,B 0,C 180,E1 -4590.768,E2 -4590.768} C_VEL
LIN {X 0,Y 524.069,Z 164.708,A -85,B 0,C 180,E1 -4593.075,E2 -4593.075} C_VEL
LIN {X 0,Y 524.05,Z 164.705,A -85,B 0,C 180,E1 -4596.159,E2 -4596.159} C_VEL
LIN {X 0,Y 523.997,Z 164.713,A -85,B 0,C 180,E1 -4599.262,E2 -4599.262} C_VEL
LIN {X 0,Y 524,Z 164.71,A -85,B 0,C 180,E1 -4601.74,E2 -4601.74} C_VEL
LIN {X 0,Y 523.99,Z 164.714,A -85,B 0,C 180,E1 -4605.053,E2 -4605.053} C_VEL
LIN {X 0,Y 523.96,Z 164.717,A -85,B 0,C 180,E1 -4607.969,E2 -4607.969} C_VEL
LIN {X 0,Y 523.968,Z 164.721,A -85,B 0,C 180,E1 -4610.41,E2 -4610.41} C_VEL
LIN {X 0,Y 523.913,Z 164.721,A -85,B 0,C 180,E1 -4612.893,E2 -4612.893} C_VEL
LIN {X 0,Y 523.948,Z 164.715,A -85,B 0,C 180,E1 -4615.418,E2 -4615.418} C_VEL
LIN {X 0,Y 523.966,Z 164.719,A -85,B 0,C 180,E1 -4617.999,E2 -4617.999} C_VEL
LIN {X 0,Y 523.948,Z 164.715,A -85,B 0,C 180,E1 -4620.856,E2 -4620.856} C_VEL
LIN {X 0,Y 523.956,Z 164.719,A -85,B 0,C 180,E1 -4623.735,E2 -4623.735} C_VEL
LIN {X 0,Y 523.917,Z 164.721,A -85,B 0,C 180,E1 -4626.404,E2 -4626.404} C_VEL
LIN {X 0,Y 523.926,Z 164.718,A -85,B 0,C 180,E1 -4629.084,E2 -4629.084} C_VEL
LIN {X 0,Y 523.967,Z 164.715,A -85,B 0,C 180,E1 -4631.312,E2 -4631.312} C_VEL
LIN {X 0,Y 523.948,Z 164.715,A -85,B 0,C 180,E1 -4634.691,E2 -4634.691} C_VEL
LIN {X 0,Y 523.95,Z 164.719,A -85,B 0,C 180,E1 -4637.882,E2 -4637.882} C_VEL
LIN {X 0,Y 523.972,Z 164.715,A -85,B 0,C 180,E1 -4639.923,E2 -4639.923} C_VEL
LIN {X 0,Y 523.905,Z 164.722,A -85,B 0,C 180,E1 -4642.868,E2 -4642.868} C_VEL
LIN {X 0,Y 523.937,Z 164.72,A -85,B 0,C 180,E1 -4645.711,E2 -4645.711} C_VEL
LIN {X 0,Y 523.918,Z 164.719,A -85,B 0,C 180,E1 -4648.456,E2 -4648.456} C_VEL
LIN {X 0,Y 523.945,Z 164.724,A -85,B 0,C 180,E1 -4651.126,E2 -4651.126} C_VEL
LIN {X 0,Y 523.977,Z 164.711,A -85,B 0,C 180,E1 -4653.98,E2 -4653.98} C_VEL
LIN {X 0,Y 523.93,Z 164.718,A -85,B 0,C 180,E1 -4656.271,E2 -4656.271} C_VEL
LIN {X 0,Y 523.941,Z 164.722,A -85,B 0,C 180,E1 -4658.767,E2 -4658.767} C_VEL
LIN {X 0,Y 523.945,Z 164.719,A -85,B 0,C 180,E1 -4661.221,E2 -4661.221} C_VEL
LIN {X 0,Y 523.931,Z 164.717,A -85,B 0,C 180,E1 -4663.639,E2 -4663.639} C_VEL
LIN {X 0,Y 523.934,Z 164.717,A -85,B 0,C 180,E1 -4666.028,E2 -4666.028} C_VEL
LIN {X 0,Y 524.005,Z 164.713,A -85,B 0,C 180,E1 -4668.394,E2 -4668.394} C_VEL
LIN {X 0,Y 523.998,Z 164.708,A -85,B 0,C 180,E1 -4671.516,E2 -4671.516} C_VEL
LIN {X 0,Y 524.076,Z 164.706,A -85,B 0,C 180,E1 -4674.614,E2 -4674.614} C_VEL
LIN {X 0,Y 524.103,Z 164.696,A -85,B 0,C 180,E1 -4677.695,E2 -4677.695} C_VEL
LIN {X 0,Y 524.118,Z 164.696,A -85,B 0,C 180,E1 -4680.769,E2 -4680.769} C_VEL
LIN {X 0,Y 524.065,Z 164.7,A -85,B 0,C 180,E1 -4683.075,E2 -4683.075} C_VEL
LIN {X 0,Y 524.038,Z 164.712,A -85,B 0,C 180,E1 -4686.16,E2 -4686.16} C_VEL
LIN {X 0,Y 523.993,Z 164.71,A -85,B 0,C 180,E1 -4689.262,E2 -4689.262} C_VEL
LIN {X 0,Y 523.997,Z 164.714,A -85,B 0,C 180,E1 -4691.74,E2 -4691.74} C_VEL
LIN {X 0,Y 523.988,Z 164.71,A -85,B 0,C 180,E1 -4695.053,E2 -4695.053} C_VEL
LIN {X 0,Y 523.958,Z 164.72,A -85,B 0,C 180,E1 -4697.97,E2 -4697.97} C_VEL
LIN {X 0,Y 523.967,Z 164.713,A -85,B 0,C 180,E1 -4700.411,E2 -4700.411} C_VEL
LIN {X 0,Y 523.91,Z 164.72,A -85,B 0,C 180,E1 -4702.894,E2 -4702.894} C_VEL
LIN {X 0,Y 523.948,Z 164.722,A -85,B 0,C 180,E1 -4705.419,E2 -4705.419} C_VEL
LIN {X 0,Y 523.953,Z 164.716,A -85,B 0,C 180,E1 -4708,E2 -4708} C_VEL
LIN {X 0,Y 523.941,Z 164.718,A -85,B 0,C 180,E1 -4710.855,E2 -4710.855} C_VEL
LIN {X 0,Y 523.955,Z 164.718,A -85,B 0,C 180,E1 -4713.735,E2 -4713.735} C_VEL
LIN {X 0,Y 523.9,Z 164.723,A -85,B 0,C 180,E1 -4716.402,E2 -4716.402} C_VEL
LIN {X 0,Y 523.919,Z 164.727,A -85,B 0,C 180,E1 -4719.085,E2 -4719.085} C_VEL
LIN {X 0,Y 523.94,Z 164.72,A -85,B 0,C 180,E1 -4722.121,E2 -4722.121} C_VEL
LIN {X 0,Y 523.921,Z 164.726,A -85,B 0,C 180,E1 -4724.688,E2 -4724.688} C_VEL
LIN {X 0,Y 524.205,Z 166.763,A -85,B 0,C 180,E1 -4726.384,E2 -4726.384} C_VEL
LIN {X 0,Y 524.621,Z 169.995,A -85,B 0,C 180,E1 -4728.608,E2 -4728.608} C_VEL
LIN {X 0,Y 524.513,Z 173.8,A -85,B 0,C 180,E1 -4731.001,E2 -4731.001} C_VEL
LIN {X 0,Y 524.288,Z 178.698,A -85,B 0,C 180,E1 -4733.857,E2 -4733.857} C_VEL
LIN {X 0,Y 524.112,Z 183.743,A -85,B 0,C 180,E1 -4736.648,E2 -4736.648} C_VEL
LIN {X 0,Y 523.997,Z 189.008,A -85,B 0,C 180,E1 -4739.359,E2 -4739.359} C_VEL
LIN {X 0,Y 523.851,Z 194.958,A -85,B 0,C 180,E1 -4742.309,E2 -4742.309} C_VEL
LIN {X 0,Y 523.743,Z 199.699,A -85,B 0,C 180,E1 -4744.571,E2 -4744.571} C_VEL
LIN {X 0,Y 523.686,Z 205.089,A -85,B 0,C 180,E1 -4747.096,E2 -4747.096} C_VEL
LIN {X 0,Y 523.613,Z 211.357,A -85,B 0,C 180,E1 -4749.977,E2 -4749.977} C_VEL
LIN {X 0,Y 523.492,Z 217.664,A -85,B 0,C 180,E1 -4752.821,E2 -4752.821} C_VEL
LIN {X 0,Y 523.44,Z 224.85,A -85,B 0,C 180,E1 -4756.015,E2 -4756.015} C_VEL
LIN {X 0,Y 523.419,Z 225.524,A -85,B 0,C 180,E1 -4756.311,E2 -4756.311} C_VEL
LIN {X 0,Y 525.386,Z 237.775,A -85,B 0,C 180,E1 -4756.659,E2 -4756.659} C_VEL
LIN {X 0,Y 525.148,Z 250.164,A -85,B 0,C 180,E1 -4757.096,E2 -4757.096} C_VEL
LIN {X 0,Y 524.855,Z 262.345,A -85,B 0,C 180,E1 -4757.694,E2 -4757.694} C_VEL
LIN {X 0,Y 524.571,Z 273.5,A -85,B 0,C 180,E1 -4758.407,E2 -4758.407} C_VEL
LIN {X 0,Y 524.344,Z 283.326,A -85,B 0,C 180,E1 -4759.185,E2 -4759.185} C_VEL
LIN {X 0,Y 524.081,Z 293.358,A -85,B 0,C 180,E1 -4760.155,E2 -4760.155} C_VEL
LIN {X 0,Y 523.854,Z 302.918,A -85,B 0,C 180,E1 -4761.319,E2 -4761.319} C_VEL
LIN {X 0,Y 523.665,Z 309.429,A -85,B 0,C 180,E1 -4762.287,E2 -4762.287} C_VEL
LIN {X 0,Y 523.525,Z 315.665,A -85,B 0,C 180,E1 -4763.418,E2 -4763.418} C_VEL
LIN {X 0,Y 523.462,Z 320.908,A -85,B 0,C 180,E1 -4764.607,E2 -4764.607} C_VEL
LIN {X 0,Y 523.441,Z 324.861,A -85,B 0,C 180,E1 -4765.765,E2 -4765.765} C_VEL
LIN {X 0,Y 523.368,Z 327.78,A -85,B 0,C 180,E1 -4766.921,E2 -4766.921} C_VEL
LIN {X 0,Y 523.275,Z 330.194,A -85,B 0,C 180,E1 -4768.461,E2 -4768.461} C_VEL
LIN {X 0,Y 523.25,Z 330.781,A -85,B 0,C 180,E1 -4769.23,E2 -4769.23} C_VEL
LIN {X 0,Y 523.25,Z 330.781,A -85,B 0,C 180,E1 -4770.77,E2 -4770.77} C_VEL
LIN {X 0,Y 523.275,Z 330.194,A -85,B 0,C 180,E1 -4771.539,E2 -4771.539} C_VEL
LIN {X 0,Y 523.368,Z 327.78,A -85,B 0,C 180,E1 -4773.079,E2 -4773.079} C_VEL
LIN {X 0,Y 523.441,Z 324.861,A -85,B 0,C 180,E1 -4774.235,E2 -4774.235} C_VEL
LIN {X 0,Y 523.462,Z 320.908,A -85,B 0,C 180,E1 -4775.393,E2 -4775.393} C_VEL
LIN {X 0,Y 523.517,Z 315.703,A -85,B 0,C 180,E1 -4776.574,E2 -4776.574} C_VEL
LIN {X 0,Y 523.665,Z 309.429,A -85,B 0,C 180,E1 -4777.713,E2 -4777.713} C_VEL
LIN {X 0,Y 523.863,Z 301.499,A -85,B 0,C 180,E1 -4778.875,E2 -4778.875} C_VEL
LIN {X 0,Y 524.081,Z 293.358,A -85,B 0,C 180,E1 -4779.845,E2 -4779.845} C_VEL
LIN {X 0,Y 524.337,Z 283.326,A -85,B 0,C 180,E1 -4780.816,E2 -4780.816} C_VEL
LIN {X 0,Y 524.61,Z 273.5,A -85,B 0,C 180,E1 -4781.592,E2 -4781.592} C_VEL
LIN {X 0,Y 524.816,Z 263.46,A -85,B 0,C 180,E1 -4782.24,E2 -4782.24} C_VEL
LIN {X 0,Y 525.102,Z 251.287,A -85,B 0,C 180,E1 -4782.856,E2 -4782.856} C_VEL
LIN {X 0,Y 525.359,Z 238.649,A -85,B 0,C 180,E1 -4783.317,E2 -4783.317} C_VEL
LIN {X 0,Y 524.53,Z 232.019,A -85,B 0,C 180,E1 -4783.524,E2 -4783.524} C_VEL
LIN {X 0,Y 523.419,Z 225.524,A -85,B 0,C 180,E1 -4783.689,E2 -4783.689} C_VEL
LIN {X 0,Y 523.438,Z 221.257,A -85,B 0,C 180,E1 -4785.577,E2 -4785.577} C_VEL
LIN {X 0,Y 523.515,Z 215.868,A -85,B 0,C 180,E1 -4787.985,E2 -4787.985} C_VEL
LIN {X 0,Y 523.618,Z 210.478,A -85,B 0,C 180,E1 -4790.424,E2 -4790.424} C_VEL
LIN {X 0,Y 523.686,Z 205.089,A -85,B 0,C 180,E1 -4792.904,E2 -4792.904} C_VEL
LIN {X 0,Y 523.803,Z 198.537,A -85,B 0,C 180,E1 -4795.978,E2 -4795.978} C_VEL
LIN {X 0,Y 523.894,Z 192.526,A -85,B 0,C 180,E1 -4798.877,E2 -4798.877} C_VEL
LIN {X 0,Y 524.009,Z 187.252,A -85,B 0,C 180,E1 -4801.538,E2 -4801.538} C_VEL
LIN {X 0,Y 524.15,Z 182.039,A -85,B 0,C 180,E1 -4804.273,E2 -4804.273} C_VEL
LIN {X 0,Y 524.338,Z 176.993,A -85,B 0,C 180,E1 -4807.096,E2 -4807.096} C_VEL
LIN {X 0,Y 524.507,Z 173.731,A -85,B 0,C 180,E1 -4809.032,E2 -4809.032} C_VEL
LIN {X 0,Y 524.62,Z 169.975,A -85,B 0,C 180,E1 -4811.392,E2 -4811.392} C_VEL
LIN {X 0,Y 524.204,Z 166.753,A -85,B 0,C 180,E1 -4813.616,E2 -4813.616} C_VEL
LIN {X 0,Y 523.921,Z 164.725,A -85,B 0,C 180,E1 -4815.312,E2 -4815.312} C_VEL
LIN {X 0,Y 523.95,Z 164.722,A -85,B 0,C 180,E1 -4818.689,E2 -4818.689} C_VEL
LIN {X 0,Y 523.916,Z 164.726,A -85,B 0,C 180,E1 -4821.08,E2 -4821.08} C_VEL
LIN {X 0,Y 523.897,Z 164.722,A -85,B 0,C 180,E1 -4823.825,E2 -4823.825} C_VEL
LIN {X 0,Y 523.938,Z 164.724,A -85,B 0,C 180,E1 -4826.635,E2 -4826.635} C_VEL
LIN {X 0,Y 523.952,Z 164.715,A -85,B 0,C 180,E1 -4829.355,E2 -4829.355} C_VEL
LIN {X 0,Y 523.969,Z 164.718,A -85,B 0,C 180,E1 -4832.282,E2 -4832.282} C_VEL
LIN {X 0,Y 523.948,Z 164.722,A -85,B 0,C 180,E1 -4834.581,E2 -4834.581} C_VEL
LIN {X 0,Y 523.912,Z 164.72,A -85,B 0,C 180,E1 -4837.106,E2 -4837.106} C_VEL
LIN {X 0,Y 523.974,Z 164.715,A -85,B 0,C 180,E1 -4839.865,E2 -4839.865} C_VEL
LIN {X 0,Y 523.962,Z 164.714,A -85,B 0,C 180,E1 -4842.837,E2 -4842.837} C_VEL
LIN {X 0,Y 523.971,Z 164.712,A -85,B 0,C 180,E1 -4845.235,E2 -4845.235} C_VEL
LIN {X 0,Y 524.007,Z 164.711,A -85,B 0,C 180,E1 -4848.394,E2 -4848.394} C_VEL
LIN {X 0,Y 523.998,Z 164.712,A -85,B 0,C 180,E1 -4851.516,E2 -4851.516} C_VEL
LIN {X 0,Y 524.075,Z 164.699,A -85,B 0,C 180,E1 -4854.613,E2 -4854.613} C_VEL
LIN {X 0,Y 524.103,Z 164.704,A -85,B 0,C 180,E1 -4857.694,E2 -4857.694} C_VEL
LIN {X 0,Y 524.117,Z 164.694,A -85,B 0,C 180,E1 -4860.768,E2 -4860.768} C_VEL
LIN {X 0,Y 524.066,Z 164.702,A -85,B 0,C 180,E1 -4863.075,E2 -4863.075} C_VEL
LIN {X 0,Y 524.039,Z 164.705,A -85,B 0,C 180,E1 -4866.159,E2 -4866.159} C_VEL
LIN {X 0,Y 523.993,Z 164.716,A -85,B 0,C 180,E1 -4869.262,E2 -4869.262} C_VEL
LIN {X 0,Y 523.996,Z 164.712,A -85,B 0,C 180,E1 -4871.739,E2 -4871.739} C_VEL
LIN {X 0,Y 523.986,Z 164.716,A -85,B 0,C 180,E1 -4875.052,E2 -4875.052} C_VEL
LIN {X 0,Y 523.957,Z 164.714,A -85,B 0,C 180,E1 -4877.969,E2 -4877.969} C_VEL
LIN {X 0,Y 523.966,Z 164.714,A -85,B 0,C 180,E1 -4880.41,E2 -4880.41} C_VEL
LIN {X 0,Y 523.91,Z 164.727,A -85,B 0,C 180,E1 -4882.893,E2 -4882.893} C_VEL
LIN {X 0,Y 523.945,Z 164.717,A -85,B 0,C 180,E1 -4885.419,E2 -4885.419} C_VEL
LIN {X 0,Y 523.963,Z 164.713,A -85,B 0,C 180,E1 -4887.999,E2 -4887.999} C_VEL
LIN {X 0,Y 523.943,Z 164.723,A -85,B 0,C 180,E1 -4890.856,E2 -4890.856} C_VEL
LIN {X 0,Y 523.954,Z 164.714,A -85,B 0,C 180,E1 -4893.735,E2 -4893.735} C_VEL
LIN {X 0,Y 523.916,Z 164.725,A -85,B 0,C 180,E1 -4896.404,E2 -4896.404} C_VEL
LIN {X 0,Y 523.925,Z 164.719,A -85,B 0,C 180,E1 -4899.084,E2 -4899.084} C_VEL
LIN {X 0,Y 523.966,Z 164.713,A -85,B 0,C 180,E1 -4901.312,E2 -4901.312} C_VEL
LIN {X 0,Y 523.95,Z 164.719,A -85,B 0,C 180,E1 -4904.691,E2 -4904.691} C_VEL
LIN {X 0,Y 523.911,Z 164.721,A -85,B 0,C 180,E1 -4906.91,E2 -4906.91} C_VEL
LIN {X 0,Y 523.246,Z 164.803,A -85,B 0,C 180,E1 -4907.551,E2 -4907.551} C_VEL
LIN {X 0,Y 520.404,Z 165.165,A -85,B 0,C 180,E1 -4908.593,E2 -4908.593} C_VEL
LIN {X 0,Y 517.999,Z 165.47,A -85,B 0,C 180,E1 -4909.432,E2 -4909.432} C_VEL
LIN {X 0,Y 516.962,Z 165.595,A -85,B 0,C 180,E1 -4910.08,E2 -4910.08} C_VEL
LIN {X 0,Y 516.876,Z 165.603,A -85,B 0,C 180,E1 -4910.299,E2 -4910.299} C_VEL
LIN {X 0,Y 516.88,Z 165.596,A -85,B 0,C 180,E1 -4913.342,E2 -4913.342} C_VEL
LIN {X 0,Y 516.907,Z 165.599,A -85,B 0,C 180,E1 -4916.121,E2 -4916.121} C_VEL
LIN {X 0,Y 516.889,Z 165.594,A -85,B 0,C 180,E1 -4918.935,E2 -4918.935} C_VEL
LIN {X 0,Y 516.92,Z 165.595,A -85,B 0,C 180,E1 -4921.585,E2 -4921.585} C_VEL
LIN {X 0,Y 516.927,Z 165.592,A -85,B 0,C 180,E1 -4924.211,E2 -4924.211} C_VEL
LIN {X 0,Y 516.868,Z 165.597,A -85,B 0,C 180,E1 -4926.777,E2 -4926.777} C_VEL
LIN {X 0,Y 516.935,Z 165.596,A -85,B 0,C 180,E1 -4929.732,E2 -4929.732} C_VEL
LIN {X 0,Y 516.925,Z 165.592,A -85,B 0,C 180,E1 -4932.596,E2 -4932.596} C_VEL
LIN {X 0,Y 516.947,Z 165.592,A -85,B 0,C 180,E1 -4935.031,E2 -4935.031} C_VEL
LIN {X 0,Y 516.962,Z 165.587,A -85,B 0,C 180,E1 -4938.234,E2 -4938.234} C_VEL
LIN {X 0,Y 516.967,Z 165.592,A -85,B 0,C 180,E1 -4941.4,E2 -4941.4} C_VEL
LIN {X 0,Y 517.013,Z 165.582,A -85,B 0,C 180,E1 -4943.757,E2 -4943.757} C_VEL
LIN {X 0,Y 517.083,Z 165.573,A -85,B 0,C 180,E1 -4947.663,E2 -4947.663} C_VEL
LIN {X 0,Y 517.091,Z 165.576,A -85,B 0,C 180,E1 -4950.779,E2 -4950.779} C_VEL
LIN {X 0,Y 517.01,Z 165.587,A -85,B 0,C 180,E1 -4953.117,E2 -4953.117} C_VEL
LIN {X 0,Y 517.013,Z 165.582,A -85,B 0,C 180,E1 -4956.243,E2 -4956.243} C_VEL
LIN {X 0,Y 516.951,Z 165.59,A -85,B 0,C 180,E1 -4959.389,E2 -4959.389} C_VEL
LIN {X 0,Y 516.949,Z 165.589,A -85,B 0,C 180,E1 -4961.807,E2 -4961.807} C_VEL
LIN {X 0,Y 516.943,Z 165.591,A -85,B 0,C 180,E1 -4965.147,E2 -4965.147} C_VEL
LIN {X 0,Y 516.922,Z 165.597,A -85,B 0,C 180,E1 -4968.222,E2 -4968.222} C_VEL
LIN {X 0,Y 516.908,Z 165.596,A -85,B 0,C 180,E1 -4970.701,E2 -4970.701} C_VEL
LIN {X 0,Y 516.907,Z 165.598,A -85,B 0,C 180,E1 -4974.072,E2 -4974.072} C_VEL
LIN {X 0,Y 516.922,Z 165.593,A -85,B 0,C 180,E1 -4976.658,E2 -4976.658} C_VEL
LIN {X 0,Y 516.92,Z 165.592,A -85,B 0,C 180,E1 -4979.526,E2 -4979.526} C_VEL
LIN {X 0,Y 516.896,Z 165.595,A -85,B 0,C 180,E1 -4982.544,E2 -4982.544} C_VEL
LIN {X 0,Y 516.878,Z 165.597,A -85,B 0,C 180,E1 -4985.332,E2 -4985.332} C_VEL
LIN {X 0,Y 516.876,Z 165.604,A -85,B 0,C 180,E1 -4987.943,E2 -4987.943} C_VEL
LIN {X 0,Y 516.898,Z 165.593,A -85,B 0,C 180,E1 -4990.739,E2 -4990.739} C_VEL
LIN {X 0,Y 516.876,Z 165.601,A -85,B 0,C 180,E1 -4993.903,E2 -4993.903} C_VEL
LIN {X 0,Y 516.876,Z 165.598,A -85,B 0,C 180,E1 -4996.107,E2 -4996.107} C_VEL
LIN {X 0,Y 516.898,Z 165.598,A -85,B 0,C 180,E1 -4999.26,E2 -4999.26} C_VEL
LIN {X 0,Y 516.858,Z 165.598,A -85,B 0,C 180,E1 -5002.274,E2 -5002.274} C_VEL
LIN {X 0,Y 516.888,Z 165.6,A -85,B 0,C 180,E1 -5005.176,E2 -5005.176} C_VEL
LIN {X 0,Y 516.87,Z 165.597,A -85,B 0,C 180,E1 -5007.975,E2 -5007.975} C_VEL
LIN {X 0,Y 516.929,Z 165.591,A -85,B 0,C 180,E1 -5010.697,E2 -5010.697} C_VEL
LIN {X 0,Y 516.936,Z 165.589,A -85,B 0,C 180,E1 -5013.804,E2 -5013.804} C_VEL
LIN {X 0,Y 516.865,Z 165.603,A -85,B 0,C 180,E1 -5016.777,E2 -5016.777} C_VEL
LIN {X 0,Y 516.933,Z 165.589,A -85,B 0,C 180,E1 -5019.732,E2 -5019.732} C_VEL
LIN {X 0,Y 516.922,Z 165.595,A -85,B 0,C 180,E1 -5022.596,E2 -5022.596} C_VEL
LIN {X 0,Y 516.935,Z 165.593,A -85,B 0,C 180,E1 -5025.03,E2 -5025.03} C_VEL
LIN {X 0,Y 516.959,Z 165.588,A -85,B 0,C 180,E1 -5028.234,E2 -5028.234} C_VEL
LIN {X 0,Y 516.963,Z 165.585,A -85,B 0,C 180,E1 -5031.4,E2 -5031.4} C_VEL
LIN {X 0,Y 517.003,Z 165.581,A -85,B 0,C 180,E1 -5033.757,E2 -5033.757} C_VEL
LIN {X 0,Y 517.075,Z 165.572,A -85,B 0,C 180,E1 -5037.664,E2 -5037.664} C_VEL
LIN {X 0,Y 517.088,Z 165.572,A -85,B 0,C 180,E1 -5040.779,E2 -5040.779} C_VEL
LIN {X 0,Y 517.006,Z 165.58,A -85,B 0,C 180,E1 -5043.117,E2 -5043.117} C_VEL
LIN {X 0,Y 517.002,Z 165.587,A -85,B 0,C 180,E1 -5046.244,E2 -5046.244} C_VEL
LIN {X 0,Y 516.948,Z 165.588,A -85,B 0,C 180,E1 -5049.39,E2 -5049.39} C_VEL
LIN {X 0,Y 516.947,Z 165.594,A -85,B 0,C 180,E1 -5051.808,E2 -5051.808} C_VEL
LIN {X 0,Y 516.939,Z 165.589,A -85,B 0,C 180,E1 -5055.147,E2 -5055.147} C_VEL
LIN {X 0,Y 516.919,Z 165.593,A -85,B 0,C 180,E1 -5058.223,E2 -5058.223} C_VEL
LIN {X 0,Y 516.907,Z 165.592,A -85,B 0,C 180,E1 -5060.702,E2 -5060.702} C_VEL
LIN {X 0,Y 516.907,Z 165.594,A -85,B 0,C 180,E1 -5064.073,E2 -5064.073} C_VEL
LIN {X 0,Y 516.918,Z 165.591,A -85,B 0,C 180,E1 -5066.659,E2 -5066.659} C_VEL
LIN {X 0,Y 516.906,Z 165.6,A -85,B 0,C 180,E1 -5069.524,E2 -5069.524} C_VEL
LIN {X 0,Y 516.892,Z 165.594,A -85,B 0,C 180,E1 -5072.544,E2 -5072.544} C_VEL
LIN {X 0,Y 516.863,Z 165.606,A -85,B 0,C 180,E1 -5075.33,E2 -5075.33} C_VEL
LIN {X 0,Y 516.877,Z 165.599,A -85,B 0,C 180,E1 -5077.944,E2 -5077.944} C_VEL
LIN {X 0,Y 516.879,Z 165.603,A -85,B 0,C 180,E1 -5080.743,E2 -5080.743} C_VEL
LIN {X 0,Y 516.879,Z 165.603,A -85,B 0,C 180,E1 -5083.904,E2 -5083.904} C_VEL
LIN {X 0,Y 516.956,Z 166.167,A -85,B 0,C 180,E1 -5085.015,E2 -5085.015} C_VEL
LIN {X 0,Y 517.406,Z 169.191,A -85,B 0,C 180,E1 -5087.223,E2 -5087.223} C_VEL
LIN {X 0,Y 517.589,Z 172.317,A -85,B 0,C 180,E1 -5089.326,E2 -5089.326} C_VEL
LIN {X 0,Y 517.409,Z 177.159,A -85,B 0,C 180,E1 -5092.322,E2 -5092.322} C_VEL
LIN {X 0,Y 517.159,Z 182.156,A -85,B 0,C 180,E1 -5095.197,E2 -5095.197} C_VEL
LIN {X 0,Y 517.014,Z 187.329,A -85,B 0,C 180,E1 -5097.985,E2 -5097.985} C_VEL
LIN {X 0,Y 516.911,Z 192.592,A -85,B 0,C 180,E1 -5100.695,E2 -5100.695} C_VEL
LIN {X 0,Y 516.742,Z 198.971,A -85,B 0,C 180,E1 -5103.85,E2 -5103.85} C_VEL
LIN {X 0,Y 516.609,Z 205.089,A -85,B 0,C 180,E1 -5106.764,E2 -5106.764} C_VEL
LIN {X 0,Y 516.55,Z 211.702,A -85,B 0,C 180,E1 -5109.85,E2 -5109.85} C_VEL
LIN {X 0,Y 516.43,Z 217.664,A -85,B 0,C 180,E1 -5112.579,E2 -5112.579} C_VEL
LIN {X 0,Y 516.356,Z 224.85,A -85,B 0,C 180,E1 -5115.819,E2 -5115.819} C_VEL
LIN {X 0,Y 516.375,Z 225.524,A -85,B 0,C 180,E1 -5116.121,E2 -5116.121} C_VEL
LIN {X 0,Y 518.45,Z 237.759,A -85,B 0,C 180,E1 -5116.477,E2 -5116.477} C_VEL
LIN {X 0,Y 518.225,Z 250.165,A -85,B 0,C 180,E1 -5116.92,E2 -5116.92} C_VEL
LIN {X 0,Y 517.908,Z 262.463,A -85,B 0,C 180,E1 -5117.534,E2 -5117.534} C_VEL
LIN {X 0,Y 517.66,Z 271.708,A -85,B 0,C 180,E1 -5118.118,E2 -5118.118} C_VEL
LIN {X 0,Y 517.383,Z 282.188,A -85,B 0,C 180,E1 -5118.938,E2 -5118.938} C_VEL
LIN {X 0,Y 517.07,Z 291.465,A -85,B 0,C 180,E1 -5119.823,E2 -5119.823} C_VEL
LIN {X 0,Y 516.874,Z 299.98,A -85,B 0,C 180,E1 -5120.807,E2 -5120.807} C_VEL
LIN {X 0,Y 516.641,Z 308.254,A -85,B 0,C 180,E1 -5121.985,E2 -5121.985} C_VEL
LIN {X 0,Y 516.482,Z 315.033,A -85,B 0,C 180,E1 -5123.199,E2 -5123.199} C_VEL
LIN {X 0,Y 516.449,Z 319.36,A -85,B 0,C 180,E1 -5124.142,E2 -5124.142} C_VEL
LIN {X 0,Y 516.271,Z 323.65,A -85,B 0,C 180,E1 -5125.315,E2 -5125.315} C_VEL
LIN {X 0,Y 516.355,Z 325.974,A -85,B 0,C 180,E1 -5126.098,E2 -5126.098} C_VEL
LIN {X 0,Y 516.283,Z 327.777,A -85,B 0,C 180,E1 -5126.879,E2 -5126.879} C_VEL
LIN {X 0,Y 516.192,Z 330.195,A -85,B 0,C 180,E1 -5128.44,E2 -5128.44} C_VEL
LIN {X 0,Y 516.16,Z 330.78,A -85,B 0,C 180,E1 -5129.22,E2 -5129.22} C_VEL
LIN {X 0,Y 516.16,Z 330.78,A -85,B 0,C 180,E1 -5130.78,E2 -5130.78} C_VEL
LIN {X 0,Y 516.192,Z 330.195,A -85,B 0,C 180,E1 -5131.56,E2 -5131.56} C_VEL
LIN {X 0,Y 516.283,Z 327.777,A -85,B 0,C 180,E1 -5133.121,E2 -5133.121} C_VEL
LIN {X 0,Y 516.343,Z 324.858,A -85,B 0,C 180,E1 -5134.293,E2 -5134.293} C_VEL
LIN {X 0,Y 516.403,Z 320.904,A -85,B 0,C 180,E1 -5135.467,E2 -5135.467} C_VEL
LIN {X 0,Y 516.444,Z 316.132,A -85,B 0,C 180,E1 -5136.575,E2 -5136.575} C_VEL
LIN {X 0,Y 516.563,Z 310.574,A -85,B 0,C 180,E1 -5137.623,E2 -5137.623} C_VEL
LIN {X 0,Y 516.755,Z 304.284,A -85,B 0,C 180,E1 -5138.604,E2 -5138.604} C_VEL
LIN {X 0,Y 516.956,Z 296.738,A -85,B 0,C 180,E1 -5139.586,E2 -5139.586} C_VEL
LIN {X 0,Y 517.242,Z 287.626,A -85,B 0,C 180,E1 -5140.569,E2 -5140.569} C_VEL
LIN {X 0,Y 517.558,Z 276.189,A -85,B 0,C 180,E1 -5141.554,E2 -5141.554} C_VEL
LIN {X 0,Y 517.744,Z 266.608,A -85,B 0,C 180,E1 -5142.217,E2 -5142.217} C_VEL
LIN {X 0,Y 518.031,Z 255.408,A -85,B 0,C 180,E1 -5142.835,E2 -5142.835} C_VEL
LIN {X 0,Y 518.306,Z 245.064,A -85,B 0,C 180,E1 -5143.277,E2 -5143.277} C_VEL
LIN {X 0,Y 518.241,Z 236.558,A -85,B 0,C 180,E1 -5143.563,E2 -5143.563} C_VEL
LIN {X 0,Y 516.375,Z 225.524,A -85,B 0,C 180,E1 -5143.879,E2 -5143.879} C_VEL
LIN {X 0,Y 516.369,Z 219.461,A -85,B 0,C 180,E1 -5146.608,E2 -5146.608} C_VEL
LIN {X 0,Y 516.461,Z 214.071,A -85,B 0,C 180,E1 -5149.062,E2 -5149.062} C_VEL
LIN {X 0,Y 516.558,Z 208.682,A -85,B 0,C 180,E1 -5151.552,E2 -5151.552} C_VEL
LIN {X 0,Y 516.671,Z 202.827,A -85,B 0,C 180,E1 -5154.305,E2 -5154.305} C_VEL
LIN {X 0,Y 516.806,Z 196.1,A -85,B 0,C 180,E1 -5157.539,E2 -5157.539} C_VEL
LIN {X 0,Y 516.932,Z 190.838,A -85,B 0,C 180,E1 -5160.201,E2 -5160.201} C_VEL
LIN {X 0,Y 517.052,Z 185.575,A -85,B 0,C 180,E1 -5162.935,E2 -5162.935} C_VEL
LIN {X 0,Y 517.215,Z 180.453,A -85,B 0,C 180,E1 -5165.752,E2 -5165.752} C_VEL
LIN {X 0,Y 517.483,Z 175.512,A -85,B 0,C 180,E1 -5168.662,E2 -5168.662} C_VEL
LIN {X 0,Y 517.607,Z 170.758,A -85,B 0,C 180,E1 -5171.687,E2 -5171.687} C_VEL
LIN {X 0,Y 517.166,Z 167.588,A -85,B 0,C 180,E1 -5173.925,E2 -5173.925} C_VEL
LIN {X 0,Y 516.956,Z 166.12,A -85,B 0,C 180,E1 -5175.013,E2 -5175.013} C_VEL
LIN {X 0,Y 516.879,Z 165.601,A -85,B 0,C 180,E1 -5176.106,E2 -5176.106} C_VEL
LIN {X 0,Y 516.879,Z 165.602,A -85,B 0,C 180,E1 -5179.257,E2 -5179.257} C_VEL
LIN {X 0,Y 516.86,Z 165.602,A -85,B 0,C 180,E1 -5182.274,E2 -5182.274} C_VEL
LIN {X 0,Y 516.88,Z 165.599,A -85,B 0,C 180,E1 -5185.175,E2 -5185.175} C_VEL
LIN {X 0,Y 516.87,Z 165.597,A -85,B 0,C 180,E1 -5187.974,E2 -5187.974} C_VEL
LIN {X 0,Y 516.917,Z 165.598,A -85,B 0,C 180,E1 -5190.695,E2 -5190.695} C_VEL
LIN {X 0,Y 516.937,Z 165.589,A -85,B 0,C 180,E1 -5193.804,E2 -5193.804} C_VEL
LIN {X 0,Y 516.868,Z 165.6,A -85,B 0,C 180,E1 -5196.776,E2 -5196.776} C_VEL
LIN {X 0,Y 516.934,Z 165.59,A -85,B 0,C 180,E1 -5199.731,E2 -5199.731} C_VEL
LIN {X 0,Y 516.916,Z 165.594,A -85,B 0,C 180,E1 -5202.595,E2 -5202.595} C_VEL
LIN {X 0,Y 516.937,Z 165.588,A -85,B 0,C 180,E1 -5205.03,E2 -5205.03} C_VEL
LIN {X 0,Y 516.96,Z 165.591,A -85,B 0,C 180,E1 -5208.233,E2 -5208.233} C_VEL
LIN {X 0,Y 516.963,Z 165.587,A -85,B 0,C 180,E1 -5211.399,E2 -5211.399} C_VEL
LIN {X 0,Y 517.002,Z 165.587,A -85,B 0,C 180,E1 -5213.756,E2 -5213.756} C_VEL
LIN {X 0,Y 517.076,Z 165.578,A -85,B 0,C 180,E1 -5217.663,E2 -5217.663} C_VEL
LIN {X 0,Y 517.087,Z 165.57,A -85,B 0,C 180,E1 -5220.778,E2 -5220.778} C_VEL
LIN {X 0,Y 517.007,Z 165.582,A -85,B 0,C 180,E1 -5223.117,E2 -5223.117} C_VEL
LIN {X 0,Y 517.003,Z 165.581,A -85,B 0,C 180,E1 -5226.243,E2 -5226.243} C_VEL
LIN {X 0,Y 516.947,Z 165.596,A -85,B 0,C 180,E1 -5229.389,E2 -5229.389} C_VEL
LIN {X 0,Y 516.945,Z 165.59,A -85,B 0,C 180,E1 -5231.807,E2 -5231.807} C_VEL
LIN {X 0,Y 516.937,Z 165.596,A -85,B 0,C 180,E1 -5235.146,E2 -5235.146} C_VEL
LIN {X 0,Y 516.918,Z 165.59,A -85,B 0,C 180,E1 -5238.222,E2 -5238.222} C_VEL
LIN {X 0,Y 516.906,Z 165.596,A -85,B 0,C 180,E1 -5240.701,E2 -5240.701} C_VEL
LIN {X 0,Y 516.904,Z 165.592,A -85,B 0,C 180,E1 -5244.072,E2 -5244.072} C_VEL
LIN {X 0,Y 516.919,Z 165.596,A -85,B 0,C 180,E1 -5246.658,E2 -5246.658} C_VEL
LIN {X 0,Y 516.918,Z 165.591,A -85,B 0,C 180,E1 -5249.526,E2 -5249.526} C_VEL
LIN {X 0,Y 516.891,Z 165.6,A -85,B 0,C 180,E1 -5252.544,E2 -5252.544} C_VEL
LIN {X 0,Y 516.876,Z 165.597,A -85,B 0,C 180,E1 -5255.332,E2 -5255.332} C_VEL
LIN {X 0,Y 516.875,Z 165.597,A -85,B 0,C 180,E1 -5257.943,E2 -5257.943} C_VEL
LIN {X 0,Y 516.898,Z 165.598,A -85,B 0,C 180,E1 -5260.74,E2 -5260.74} C_VEL
LIN {X 0,Y 516.876,Z 165.598,A -85,B 0,C 180,E1 -5263.903,E2 -5263.903} C_VEL
LIN {X 0,Y 516.875,Z 165.602,A -85,B 0,C 180,E1 -5266.107,E2 -5266.107} C_VEL
LIN {X 0,Y 516.911,Z 165.598,A -85,B 0,C 180,E1 -5268.398,E2 -5268.398} C_VEL
LIN {X 0,Y 516.876,Z 165.603,A -85,B 0,C 180,E1 -5270.299,E2 -5270.299} C_VEL
LIN {X 0,Y 516.207,Z 165.681,A -85,B 0,C 180,E1 -5270.949,E2 -5270.949} C_VEL
LIN {X 0,Y 513.362,Z 166.04,A -85,B 0,C 180,E1 -5272.005,E2 -5272.005} C_VEL
LIN {X 0,Y 510.955,Z 166.34,A -85,B 0,C 180,E1 -5272.855,E2 -5272.855} C_VEL
LIN {X 0,Y 509.915,Z 166.466,A -85,B 0,C 180,E1 -5273.512,E2 -5273.512} C_VEL
LIN {X 0,Y 509.826,Z 166.476,A -85,B 0,C 180,E1 -5273.734,E2 -5273.734} C_VEL
LIN {X 0,Y 509.858,Z 166.472,A -85,B 0,C 180,E1 -5276.54,E2 -5276.54} C_VEL
LIN {X 0,Y 509.846,Z 166.473,A -85,B 0,C 180,E1 -5279.335,E2 -5279.335} C_VEL
LIN {X 0,Y 509.89,Z 166.471,A -85,B 0,C 180,E1 -5282.055,E2 -5282.055} C_VEL
LIN {X 0,Y 509.873,Z 166.468,A -85,B 0,C 180,E1 -5284.704,E2 -5284.704} C_VEL
LIN {X 0,Y 509.832,Z 166.479,A -85,B 0,C 180,E1 -5287.455,E2 -5287.455} C_VEL
LIN {X 0,Y 509.913,Z 166.47,A -85,B 0,C 180,E1 -5289.845,E2 -5289.845} C_VEL
LIN {X 0,Y 509.881,Z 166.473,A -85,B 0,C 180,E1 -5293.175,E2 -5293.175} C_VEL
LIN {X 0,Y 509.87,Z 166.476,A -85,B 0,C 180,E1 -5295.635,E2 -5295.635} C_VEL
LIN {X 0,Y 509.91,Z 166.468,A -85,B 0,C 180,E1 -5298.875,E2 -5298.875} C_VEL
LIN {X 0,Y 509.948,Z 166.461,A -85,B 0,C 180,E1 -5302.079,E2 -5302.079} C_VEL
LIN {X 0,Y 509.983,Z 166.457,A -85,B 0,C 180,E1 -5304.464,E2 -5304.464} C_VEL
LIN {X 0,Y 510.053,Z 166.449,A -85,B 0,C 180,E1 -5307.631,E2 -5307.631} C_VEL
LIN {X 0,Y 510.061,Z 166.452,A -85,B 0,C 180,E1 -5310.789,E2 -5310.789} C_VEL
LIN {X 0,Y 509.953,Z 166.466,A -85,B 0,C 180,E1 -5313.16,E2 -5313.16} C_VEL
LIN {X 0,Y 509.98,Z 166.459,A -85,B 0,C 180,E1 -5316.329,E2 -5316.329} C_VEL
LIN {X 0,Y 509.913,Z 166.472,A -85,B 0,C 180,E1 -5318.72,E2 -5318.72} C_VEL
LIN {X 0,Y 509.901,Z 166.467,A -85,B 0,C 180,E1 -5321.932,E2 -5321.932} C_VEL
LIN {X 0,Y 509.89,Z 166.469,A -85,B 0,C 180,E1 -5325.242,E2 -5325.242} C_VEL
LIN {X 0,Y 509.885,Z 166.471,A -85,B 0,C 180,E1 -5328.001,E2 -5328.001} C_VEL
LIN {X 0,Y 509.846,Z 166.473,A -85,B 0,C 180,E1 -5331.002,E2 -5331.002} C_VEL
LIN {X 0,Y 509.832,Z 166.474,A -85,B 0,C 180,E1 -5333.563,E2 -5333.563} C_VEL
LIN {X 0,Y 509.907,Z 166.47,A -85,B 0,C 180,E1 -5336.379,E2 -5336.379} C_VEL
LIN {X 0,Y 509.881,Z 166.468,A -85,B 0,C 180,E1 -5338.843,E2 -5338.843} C_VEL
LIN {X 0,Y 509.822,Z 166.477,A -85,B 0,C 180,E1 -5341.589,E2 -5341.589} C_VEL
LIN {X 0,Y 509.849,Z 166.474,A -85,B 0,C 180,E1 -5344.413,E2 -5344.413} C_VEL
LIN {X 0,Y 509.814,Z 166.477,A -85,B 0,C 180,E1 -5347.34,E2 -5347.34} C_VEL
LIN {X 0,Y 509.856,Z 166.472,A -85,B 0,C 180,E1 -5350.38,E2 -5350.38} C_VEL
LIN {X 0,Y 509.817,Z 166.476,A -85,B 0,C 180,E1 -5353.062,E2 -5353.062} C_VEL
LIN {X 0,Y 509.825,Z 166.481,A -85,B 0,C 180,E1 -5355.792,E2 -5355.792} C_VEL
LIN {X 0,Y 509.859,Z 166.47,A -85,B 0,C 180,E1 -5358.576,E2 -5358.576} C_VEL
LIN {X 0,Y 509.846,Z 166.476,A -85,B 0,C 180,E1 -5361.786,E2 -5361.786} C_VEL
LIN {X 0,Y 509.839,Z 166.473,A -85,B 0,C 180,E1 -5364.623,E2 -5364.623} C_VEL
LIN {X 0,Y 509.856,Z 166.476,A -85,B 0,C 180,E1 -5367.481,E2 -5367.481} C_VEL
LIN {X 0,Y 509.875,Z 166.468,A -85,B 0,C 180,E1 -5370.269,E2 -5370.269} C_VEL
LIN {X 0,Y 509.879,Z 166.474,A -85,B 0,C 180,E1 -5372.945,E2 -5372.945} C_VEL
LIN {X 0,Y 509.863,Z 166.471,A -85,B 0,C 180,E1 -5375.574,E2 -5375.574} C_VEL
LIN {X 0,Y 509.844,Z 166.48,A -85,B 0,C 180,E1 -5378.999,E2 -5378.999} C_VEL
LIN {X 0,Y 509.882,Z 166.467,A -85,B 0,C 180,E1 -5381.999,E2 -5381.999} C_VEL
LIN {X 0,Y 509.903,Z 166.473,A -85,B 0,C 180,E1 -5384.819,E2 -5384.819} C_VEL
LIN {X 0,Y 509.894,Z 166.467,A -85,B 0,C 180,E1 -5388.124,E2 -5388.124} C_VEL
LIN {X 0,Y 509.91,Z 166.464,A -85,B 0,C 180,E1 -5391.28,E2 -5391.28} C_VEL
LIN {X 0,Y 509.971,Z 166.456,A -85,B 0,C 180,E1 -5393.671,E2 -5393.671} C_VEL
LIN {X 0,Y 510.046,Z 166.447,A -85,B 0,C 180,E1 -5397.631,E2 -5397.631} C_VEL
LIN {X 0,Y 510.058,Z 166.447,A -85,B 0,C 180,E1 -5400.79,E2 -5400.79} C_VEL
LIN {X 0,Y 509.948,Z 166.459,A -85,B 0,C 180,E1 -5403.161,E2 -5403.161} C_VEL
LIN {X 0,Y 509.953,Z 166.464,A -85,B 0,C 180,E1 -5406.33,E2 -5406.33} C_VEL
LIN {X 0,Y 509.91,Z 166.465,A -85,B 0,C 180,E1 -5408.721,E2 -5408.721} C_VEL
LIN {X 0,Y 509.899,Z 166.474,A -85,B 0,C 180,E1 -5411.932,E2 -5411.932} C_VEL
LIN {X 0,Y 509.889,Z 166.467,A -85,B 0,C 180,E1 -5415.242,E2 -5415.242} C_VEL
LIN {X 0,Y 509.877,Z 166.473,A -85,B 0,C 180,E1 -5417.999,E2 -5417.999} C_VEL
LIN {X 0,Y 509.846,Z 166.472,A -85,B 0,C 180,E1 -5421.002,E2 -5421.002} C_VEL
LIN {X 0,Y 509.866,Z 166.469,A -85,B 0,C 180,E1 -5424.427,E2 -5424.427} C_VEL
LIN {X 0,Y 509.877,Z 166.47,A -85,B 0,C 180,E1 -5427.057,E2 -5427.057} C_VEL
LIN {X 0,Y 509.853,Z 166.475,A -85,B 0,C 180,E1 -5429.752,E2 -5429.752} C_VEL
LIN {X 0,Y 509.869,Z 166.47,A -85,B 0,C 180,E1 -5432.775,E2 -5432.775} C_VEL
LIN {X 0,Y 509.822,Z 166.481,A -85,B 0,C 180,E1 -5435.579,E2 -5435.579} C_VEL
LIN {X 0,Y 509.847,Z 166.475,A -85,B 0,C 180,E1 -5438.339,E2 -5438.339} C_VEL
LIN {X 0,Y 509.85,Z 166.479,A -85,B 0,C 180,E1 -5441.427,E2 -5441.427} C_VEL
LIN {X 0,Y 509.821,Z 166.482,A -85,B 0,C 180,E1 -5444.207,E2 -5444.207} C_VEL
LIN {X 0,Y 510.349,Z 169.939,A -85,B 0,C 180,E1 -5446.875,E2 -5446.875} C_VEL
LIN {X 0,Y 510.603,Z 173.327,A -85,B 0,C 180,E1 -5449.203,E2 -5449.203} C_VEL
LIN {X 0,Y 510.458,Z 177.276,A -85,B 0,C 180,E1 -5451.717,E2 -5451.717} C_VEL
LIN {X 0,Y 510.181,Z 182.258,A -85,B 0,C 180,E1 -5454.651,E2 -5454.651} C_VEL
LIN {X 0,Y 510,Z 187.338,A -85,B 0,C 180,E1 -5457.491,E2 -5457.491} C_VEL
LIN {X 0,Y 509.861,Z 192.636,A -85,B 0,C 180,E1 -5460.274,E2 -5460.274} C_VEL
LIN {X 0,Y 509.719,Z 197.851,A -85,B 0,C 180,E1 -5462.935,E2 -5462.935} C_VEL
LIN {X 0,Y 509.618,Z 203.292,A -85,B 0,C 180,E1 -5465.562,E2 -5465.562} C_VEL
LIN {X 0,Y 509.519,Z 208.682,A -85,B 0,C 180,E1 -5468.135,E2 -5468.135} C_VEL
LIN {X 0,Y 509.395,Z 214.071,A -85,B 0,C 180,E1 -5470.663,E2 -5470.663} C_VEL
LIN {X 0,Y 509.308,Z 219.461,A -85,B 0,C 180,E1 -5473.155,E2 -5473.155} C_VEL
LIN {X 0,Y 509.277,Z 225.524,A -85,B 0,C 180,E1 -5475.923,E2 -5475.923} C_VEL
LIN {X 0,Y 511.407,Z 238.18,A -85,B 0,C 180,E1 -5476.3,E2 -5476.3} C_VEL
LIN {X 0,Y 511.286,Z 251.294,A -85,B 0,C 180,E1 -5476.79,E2 -5476.79} C_VEL
LIN {X 0,Y 510.964,Z 262.467,A -85,B 0,C 180,E1 -5477.362,E2 -5477.362} C_VEL
LIN {X 0,Y 510.69,Z 272.099,A -85,B 0,C 180,E1 -5477.984,E2 -5477.984} C_VEL
LIN {X 0,Y 510.403,Z 282.181,A -85,B 0,C 180,E1 -5478.785,E2 -5478.785} C_VEL
LIN {X 0,Y 510.181,Z 289.547,A -85,B 0,C 180,E1 -5479.483,E2 -5479.483} C_VEL
LIN {X 0,Y 509.951,Z 296.734,A -85,B 0,C 180,E1 -5480.281,E2 -5480.281} C_VEL
LIN {X 0,Y 509.72,Z 304.28,A -85,B 0,C 180,E1 -5481.277,E2 -5481.277} C_VEL
LIN {X 0,Y 509.522,Z 310.569,A -85,B 0,C 180,E1 -5482.271,E2 -5482.271} C_VEL
LIN {X 0,Y 509.35,Z 316.657,A -85,B 0,C 180,E1 -5483.443,E2 -5483.443} C_VEL
LIN {X 0,Y 509.247,Z 322.386,A -85,B 0,C 180,E1 -5484.853,E2 -5484.853} C_VEL
LIN {X 0,Y 509.268,Z 325.975,A -85,B 0,C 180,E1 -5486.043,E2 -5486.043} C_VEL
LIN {X 0,Y 509.201,Z 327.775,A -85,B 0,C 180,E1 -5486.835,E2 -5486.835} C_VEL
LIN {X 0,Y 509.113,Z 330.195,A -85,B 0,C 180,E1 -5488.418,E2 -5488.418} C_VEL
LIN {X 0,Y 509.074,Z 330.78,A -85,B 0,C 180,E1 -5489.209,E2 -5489.209} C_VEL
LIN {X 0,Y 509.074,Z 330.78,A -85,B 0,C 180,E1 -5490.791,E2 -5490.791} C_VEL
LIN {X 0,Y 509.113,Z 330.195,A -85,B 0,C 180,E1 -5491.582,E2 -5491.582} C_VEL
LIN {X 0,Y 509.201,Z 327.775,A -85,B 0,C 180,E1 -5493.165,E2 -5493.165} C_VEL
LIN {X 0,Y 509.233,Z 324.854,A -85,B 0,C 180,E1 -5494.353,E2 -5494.353} C_VEL
LIN {X 0,Y 509.342,Z 320.899,A -85,B 0,C 180,E1 -5495.543,E2 -5495.543} C_VEL
LIN {X 0,Y 509.404,Z 315.277,A -85,B 0,C 180,E1 -5496.844,E2 -5496.844} C_VEL
LIN {X 0,Y 509.585,Z 308.255,A -85,B 0,C 180,E1 -5498.127,E2 -5498.127} C_VEL
LIN {X 0,Y 509.85,Z 299.975,A -85,B 0,C 180,E1 -5499.321,E2 -5499.321} C_VEL
LIN {X 0,Y 510.062,Z 291.46,A -85,B 0,C 180,E1 -5500.319,E2 -5500.319} C_VEL
LIN {X 0,Y 510.384,Z 283.313,A -85,B 0,C 180,E1 -5501.115,E2 -5501.115} C_VEL
LIN {X 0,Y 510.65,Z 274.833,A -85,B 0,C 180,E1 -5501.813,E2 -5501.813} C_VEL
LIN {X 0,Y 510.836,Z 266.107,A -85,B 0,C 180,E1 -5502.416,E2 -5502.416} C_VEL
LIN {X 0,Y 511.125,Z 255.399,A -85,B 0,C 180,E1 -5503.012,E2 -5503.012} C_VEL
LIN {X 0,Y 511.411,Z 245.055,A -85,B 0,C 180,E1 -5503.459,E2 -5503.459} C_VEL
LIN {X 0,Y 511.371,Z 237.743,A -85,B 0,C 180,E1 -5503.714,E2 -5503.714} C_VEL
LIN {X 0,Y 509.419,Z 226.61,A -85,B 0,C 180,E1 -5504.047,E2 -5504.047} C_VEL
LIN {X 0,Y 509.277,Z 225.524,A -85,B 0,C 180,E1 -5504.077,E2 -5504.077} C_VEL
LIN {X 0,Y 509.308,Z 219.461,A -85,B 0,C 180,E1 -5506.845,E2 -5506.845} C_VEL
LIN {X 0,Y 509.395,Z 214.071,A -85,B 0,C 180,E1 -5509.337,E2 -5509.337} C_VEL
LIN {X 0,Y 509.519,Z 208.682,A -85,B 0,C 180,E1 -5511.865,E2 -5511.865} C_VEL
LIN {X 0,Y 509.625,Z 203.226,A -85,B 0,C 180,E1 -5514.47,E2 -5514.47} C_VEL
LIN {X 0,Y 509.719,Z 197.851,A -85,B 0,C 180,E1 -5517.065,E2 -5517.065} C_VEL
LIN {X 0,Y 509.861,Z 192.589,A -85,B 0,C 180,E1 -5519.75,E2 -5519.75} C_VEL
LIN {X 0,Y 510.012,Z 186.798,A -85,B 0,C 180,E1 -5522.798,E2 -5522.798} C_VEL
LIN {X 0,Y 510.196,Z 181.718,A -85,B 0,C 180,E1 -5525.636,E2 -5525.636} C_VEL
LIN {X 0,Y 510.444,Z 177.247,A -85,B 0,C 180,E1 -5528.297,E2 -5528.297} C_VEL
LIN {X 0,Y 510.6,Z 173.281,A -85,B 0,C 180,E1 -5530.796,E2 -5530.796} C_VEL
LIN {X 0,Y 510.349,Z 169.937,A -85,B 0,C 180,E1 -5533.125,E2 -5533.125} C_VEL
LIN {X 0,Y 509.821,Z 166.481,A -85,B 0,C 180,E1 -5535.793,E2 -5535.793} C_VEL
LIN {X 0,Y 509.85,Z 166.478,A -85,B 0,C 180,E1 -5538.573,E2 -5538.573} C_VEL
LIN {X 0,Y 509.848,Z 166.474,A -85,B 0,C 180,E1 -5541.786,E2 -5541.786} C_VEL
LIN {X 0,Y 509.826,Z 166.481,A -85,B 0,C 180,E1 -5544.621,E2 -5544.621} C_VEL
LIN {X 0,Y 509.858,Z 166.47,A -85,B 0,C 180,E1 -5547.48,E2 -5547.48} C_VEL
LIN {X 0,Y 509.855,Z 166.475,A -85,B 0,C 180,E1 -5550.273,E2 -5550.273} C_VEL
LIN {X 0,Y 509.877,Z 166.47,A -85,B 0,C 180,E1 -5552.943,E2 -5552.943} C_VEL
LIN {X 0,Y 509.866,Z 166.469,A -85,B 0,C 180,E1 -5555.573,E2 -5555.573} C_VEL
LIN {X 0,Y 509.846,Z 166.472,A -85,B 0,C 180,E1 -5558.998,E2 -5558.998} C_VEL
LIN {X 0,Y 509.877,Z 166.473,A -85,B 0,C 180,E1 -5562.001,E2 -5562.001} C_VEL
LIN {X 0,Y 509.905,Z 166.465,A -85,B 0,C 180,E1 -5564.818,E2 -5564.818} C_VEL
LIN {X 0,Y 509.895,Z 166.473,A -85,B 0,C 180,E1 -5568.123,E2 -5568.123} C_VEL
LIN {X 0,Y 509.91,Z 166.465,A -85,B 0,C 180,E1 -5571.279,E2 -5571.279} C_VEL
LIN {X 0,Y 509.953,Z 166.464,A -85,B 0,C 180,E1 -5573.67,E2 -5573.67} C_VEL
LIN {X 0,Y 510.047,Z 166.453,A -85,B 0,C 180,E1 -5577.63,E2 -5577.63} C_VEL
LIN {X 0,Y 510.048,Z 166.451,A -85,B 0,C 180,E1 -5580,E2 -5580} C_VEL
LIN {X 0,Y 510.046,Z 166.447,A -85,B 0,C 180,E1 -5582.369,E2 -5582.369} C_VEL
LIN {X 0,Y 509.971,Z 166.456,A -85,B 0,C 180,E1 -5586.329,E2 -5586.329} C_VEL
LIN {X 0,Y 509.91,Z 166.464,A -85,B 0,C 180,E1 -5588.72,E2 -5588.72} C_VEL
LIN {X 0,Y 509.897,Z 166.467,A -85,B 0,C 180,E1 -5591.931,E2 -5591.931} C_VEL
LIN {X 0,Y 509.887,Z 166.475,A -85,B 0,C 180,E1 -5595.242,E2 -5595.242} C_VEL
LIN {X 0,Y 509.882,Z 166.467,A -85,B 0,C 180,E1 -5598.001,E2 -5598.001} C_VEL
LIN {X 0,Y 509.844,Z 166.48,A -85,B 0,C 180,E1 -5601.001,E2 -5601.001} C_VEL
LIN {X 0,Y 509.863,Z 166.471,A -85,B 0,C 180,E1 -5604.426,E2 -5604.426} C_VEL
LIN {X 0,Y 509.879,Z 166.474,A -85,B 0,C 180,E1 -5607.055,E2 -5607.055} C_VEL
LIN {X 0,Y 509.874,Z 166.468,A -85,B 0,C 180,E1 -5609.749,E2 -5609.749} C_VEL
LIN {X 0,Y 509.867,Z 166.477,A -85,B 0,C 180,E1 -5612.774,E2 -5612.774} C_VEL
LIN {X 0,Y 509.836,Z 166.473,A -85,B 0,C 180,E1 -5615.581,E2 -5615.581} C_VEL
LIN {X 0,Y 509.845,Z 166.477,A -85,B 0,C 180,E1 -5618.338,E2 -5618.338} C_VEL
LIN {X 0,Y 509.859,Z 166.47,A -85,B 0,C 180,E1 -5621.424,E2 -5621.424} C_VEL
LIN {X 0,Y 509.85,Z 166.475,A -85,B 0,C 180,E1 -5624.668,E2 -5624.668} C_VEL
LIN {X 0,Y 509.853,Z 166.477,A -85,B 0,C 180,E1 -5628.103,E2 -5628.103} C_VEL
